# B&R Automation Studio project A2019059_Linka_Power_CP (part 30)

#### AtlasCopcoKomunikacia.st
```iecst
ACTION AtlasCopcoKomunikacia:

    M5_PrevodMomentu();
    M4_PrevodMomentu();
    M6_PrevodMomentu();

	//*********************************************************Skrutkovacka M5******************************************************************//
	//Vstupy z AtlasCopco do PLC//
    P2_Srobovanie.Skrutkovacka_M5.Stav_VysledokPotvrdeny:= P2_Srobovanie.PAR.M5_AtlasCopcoInputs[0].0;
    P2_Srobovanie.Skrutkovacka_M5.Stav_EmergencyStop:= P2_Srobovanie.PAR.M5_AtlasCopcoInputs[0].1;
    P2_Srobovanie.Skrutkovacka_M5.Stav_READY_to_START:= P2_Srobovanie.PAR.M5_AtlasCopcoInputs[0].2;
    P2_Srobovanie.Skrutkovacka_M5.Stav_MANUAL:= P2_Srobovanie.PAR.M5_AtlasCopcoInputs[0].3;
    P2_Srobovanie.Skrutkovacka_M5.Stav_UtahovanieUkoncene:= P2_Srobovanie.PAR.M5_AtlasCopcoInputs[0].4;
    P2_Srobovanie.Skrutkovacka_M5.Stav_VysledokUtahovania_NG:= P2_Srobovanie.PAR.M5_AtlasCopcoInputs[0].5;
    P2_Srobovanie.Skrutkovacka_M5.Stav_VysledokUtahovania_OK:= P2_Srobovanie.PAR.M5_AtlasCopcoInputs[0].6;
    P2_Srobovanie.Skrutkovacka_M5.Stav_SmerOtacania_VPRED:= P2_Srobovanie.PAR.M5_AtlasCopcoInputs[0].7;
    P2_Srobovanie.Skrutkovacka_M5.Stav_BUSY:= P2_Srobovanie.PAR.M5_AtlasCopcoInputs[0].8;
    P2_Srobovanie.Skrutkovacka_M5.Stav_ControlerSwitch_ON:= P2_Srobovanie.PAR.M5_AtlasCopcoInputs[0].9;
    P2_Srobovanie.Skrutkovacka_M5.Stav_Station_READY:= P2_Srobovanie.PAR.M5_AtlasCopcoInputs[0].10;
    P2_Srobovanie.Skrutkovacka_M5.Stav_NastrojPripojeny:= P2_Srobovanie.PAR.M5_AtlasCopcoInputs[0].11;
    P2_Srobovanie.Skrutkovacka_M5.Stav_NastrojUtahuje:= P2_Srobovanie.PAR.M5_AtlasCopcoInputs[0].12;

    //Výstupy z PLC do AtlasCopco//
    P2_Srobovanie.PAR.M5_AllasCopcoOutputs[0].0:= P2_Srobovanie.Skrutkovacka_M5.RESET_Poruchy;
    P2_Srobovanie.PAR.M5_AllasCopcoOutputs[0].1:= P2_Srobovanie.Skrutkovacka_M5.RESET_Vysledkov;
    P2_Srobovanie.PAR.M5_AllasCopcoOutputs[0].2:= P2_Srobovanie.Skrutkovacka_M5.START_Skrutkovania;
    P2_Srobovanie.PAR.M5_AllasCopcoOutputs[0].3:= P2_Srobovanie.Skrutkovacka_M5.START_Utahovania;

    //Dosiahnutý moment//
//    P2_Srobovanie.STAV.M5_DosiahnutyMoment.0:= P2_Srobovanie.PAR.M5_AtlasCopcoInputs[1].24;
//    P2_Srobovanie.STAV.M5_DosiahnutyMoment.1:= P2_Srobovanie.PAR.M5_AtlasCopcoInputs[1].25;
//    P2_Srobovanie.STAV.M5_DosiahnutyMoment.2:= P2_Srobovanie.PAR.M5_AtlasCopcoInputs[1].26;
//    P2_Srobovanie.STAV.M5_DosiahnutyMoment.3:= P2_Srobovanie.PAR.M5_AtlasCopcoInputs[1].27;
//    P2_Srobovanie.STAV.M5_DosiahnutyMoment.4:= P2_Srobovanie.PAR.M5_AtlasCopcoInputs[1].28;
//    P2_Srobovanie.STAV.M5_DosiahnutyMoment.5:= P2_Srobovanie.PAR.M5_AtlasCopcoInputs[1].29;
//    P2_Srobovanie.STAV.M5_DosiahnutyMoment.6:= P2_Srobovanie.PAR.M5_AtlasCopcoInputs[1].30;
//    P2_Srobovanie.STAV.M5_DosiahnutyMoment.7:= P2_Srobovanie.PAR.M5_AtlasCopcoInputs[1].31;
//    P2_Srobovanie.STAV.M5_DosiahnutyMoment.8:= P2_Srobovanie.PAR.M5_AtlasCopcoInputs[1].16;
//    P2_Srobovanie.STAV.M5_DosiahnutyMoment.9:= P2_Srobovanie.PAR.M5_AtlasCopcoInputs[1].17;
//    P2_Srobovanie.STAV.M5_DosiahnutyMoment.10:= P2_Srobovanie.PAR.M5_AtlasCopcoInputs[1].18;
//    P2_Srobovanie.STAV.M5_DosiahnutyMoment.11:= P2_Srobovanie.PAR.M5_AtlasCopcoInputs[1].19;
//    P2_Srobovanie.STAV.M5_DosiahnutyMoment.12:= P2_Srobovanie.PAR.M5_AtlasCopcoInputs[1].20;
//    P2_Srobovanie.STAV.M5_DosiahnutyMoment.13:= P2_Srobovanie.PAR.M5_AtlasCopcoInputs[1].21;
//    P2_Srobovanie.STAV.M5_DosiahnutyMoment.14:= P2_Srobovanie.PAR.M5_AtlasCopcoInputs[1].22;
//    P2_Srobovanie.STAV.M5_DosiahnutyMoment.15:= P2_Srobovanie.PAR.M5_AtlasCopcoInputs[1].23;
//    P2_Srobovanie.STAV.M5_DosiahnutyMoment.16:= P2_Srobovanie.PAR.M5_AtlasCopcoInputs[1].8;
//    P2_Srobovanie.STAV.M5_DosiahnutyMoment.17:= P2_Srobovanie.PAR.M5_AtlasCopcoInputs[1].9;
//    P2_Srobovanie.STAV.M5_DosiahnutyMoment.18:= P2_Srobovanie.PAR.M5_AtlasCopcoInputs[1].10;
//    P2_Srobovanie.STAV.M5_DosiahnutyMoment.19:= P2_Srobovanie.PAR.M5_AtlasCopcoInputs[1].11;
//    P2_Srobovanie.STAV.M5_DosiahnutyMoment.20:= P2_Srobovanie.PAR.M5_AtlasCopcoInputs[1].12;
//    P2_Srobovanie.STAV.M5_DosiahnutyMoment.21:= P2_Srobovanie.PAR.M5_AtlasCopcoInputs[1].13;
//    P2_Srobovanie.STAV.M5_DosiahnutyMoment.22:= P2_Srobovanie.PAR.M5_AtlasCopcoInputs[1].14;
//    P2_Srobovanie.STAV.M5_DosiahnutyMoment.23:= P2_Srobovanie.PAR.M5_AtlasCopcoInputs[1].15;
//    P2_Srobovanie.STAV.M5_DosiahnutyMoment.24:= P2_Srobovanie.PAR.M5_AtlasCopcoInputs[1].0;
//    P2_Srobovanie.STAV.M5_DosiahnutyMoment.25:= P2_Srobovanie.PAR.M5_AtlasCopcoInputs[1].1;
//    P2_Srobovanie.STAV.M5_DosiahnutyMoment.26:= P2_Srobovanie.PAR.M5_AtlasCopcoInputs[1].2;
//    P2_Srobovanie.STAV.M5_DosiahnutyMoment.27:= P2_Srobovanie.PAR.M5_AtlasCopcoInputs[1].3;
//    P2_Srobovanie.STAV.M5_DosiahnutyMoment.28:= P2_Srobovanie.PAR.M5_AtlasCopcoInputs[1].4;
//    P2_Srobovanie.STAV.M5_DosiahnutyMoment.29:= P2_Srobovanie.PAR.M5_AtlasCopcoInputs[1].5;
//    P2_Srobovanie.STAV.M5_DosiahnutyMoment.30:= P2_Srobovanie.PAR.M5_AtlasCopcoInputs[1].6;
//    P2_Srobovanie.STAV.M5_DosiahnutyMoment.31:= P2_Srobovanie.PAR.M5_AtlasCopcoInputs[1].7;
//    M5_DosiahnutyMoment_REAL:= UDINT_TO_REAL(P2_Srobovanie.STAV.M5_DosiahnutyMoment);
//    IF M5_DosiahnutyMoment_REAL > 0 THEN
//        P2_Srobovanie.STAV.M5_DosiahnutyMoment_REAL:= M5_DosiahnutyMoment_REAL/100;
//    ELSE
//        P2_Srobovanie.STAV.M5_DosiahnutyMoment_REAL:= 0.0;
//    END_IF

    M5_PrevodMomentu.AtlasAktualnyMoment:=P2_Srobovanie.PAR.M5_AtlasCopcoInputs[1];
    P2_Srobovanie.STAV.M5_DosiahnutyMoment_REAL:=M5_PrevodMomentu.AktualnyMoment;

    //Moment - Tolerancia MAX//
//    P2_Srobovanie.STAV.M5_Moment_ToleranciaMAX.0:= P2_Srobovanie.PAR.M5_AtlasCopcoInputs[3].24;
//    P2_Srobovanie.STAV.M5_Moment_ToleranciaMAX.1:= P2_Srobovanie.PAR.M5_AtlasCopcoInputs[3].25;
//    P2_Srobovanie.STAV.M5_Moment_ToleranciaMAX.2:= P2_Srobovanie.PAR.M5_AtlasCopcoInputs[3].26;
//    P2_Srobovanie.STAV.M5_Moment_ToleranciaMAX.3:= P2_Srobovanie.PAR.M5_AtlasCopcoInputs[3].27;
//    P2_Srobovanie.STAV.M5_Moment_ToleranciaMAX.4:= P2_Srobovanie.PAR.M5_AtlasCopcoInputs[3].28;
//    P2_Srobovanie.STAV.M5_Moment_ToleranciaMAX.5:= P2_Srobovanie.PAR.M5_AtlasCopcoInputs[3].29;
//    P2_Srobovanie.STAV.M5_Moment_ToleranciaMAX.6:= P2_Srobovanie.PAR.M5_AtlasCopcoInputs[3].30;
//    P2_Srobovanie.STAV.M5_Moment_ToleranciaMAX.7:= P2_Srobovanie.PAR.M5_AtlasCopcoInputs[3].31;
//    P2_Srobovanie.STAV.M5_Moment_ToleranciaMAX.8:= P2_Srobovanie.PAR.M5_AtlasCopcoInputs[3].16;
//    P2_Srobovanie.STAV.M5_Moment_ToleranciaMAX.9:= P2_Srobovanie.PAR.M5_AtlasCopcoInputs[3].17;
//    P2_Srobovanie.STAV.M5_Moment_ToleranciaMAX.10:= P2_Srobovanie.PAR.M5_AtlasCopcoInputs[3].18;
//    P2_Srobovanie.STAV.M5_Moment_ToleranciaMAX.11:= P2_Srobovanie.PAR.M5_AtlasCopcoInputs[3].19;
//    P2_Srobovanie.STAV.M5_Moment_ToleranciaMAX.12:= P2_Srobovanie.PAR.M5_AtlasCopcoInputs[3].20;
//    P2_Srobovanie.STAV.M5_Moment_ToleranciaMAX.13:= P2_Srobovanie.PAR.M5_AtlasCopcoInputs[3].21;
//    P2_Srobovanie.STAV.M5_Moment_ToleranciaMAX.14:= P2_Srobovanie.PAR.M5_AtlasCopcoInputs[3].22;
//    P2_Srobovanie.STAV.M5_Moment_ToleranciaMAX.15:= P2_Srobovanie.PAR.M5_AtlasCopcoInputs[3].23;
//    P2_Srobovanie.STAV.M5_Moment_ToleranciaMAX.16:= P2_Srobovanie.PAR.M5_AtlasCopcoInputs[3].8;
//    P2_Srobovanie.STAV.M5_Moment_ToleranciaMAX.17:= P2_Srobovanie.PAR.M5_AtlasCopcoInputs[3].9;
//    P2_Srobovanie.STAV.M5_Moment_ToleranciaMAX.18:= P2_Srobovanie.PAR.M5_AtlasCopcoInputs[3].10;
//    P2_Srobovanie.STAV.M5_Moment_ToleranciaMAX.19:= P2_Srobovanie.PAR.M5_AtlasCopcoInputs[3].11;
//    P2_Srobovanie.STAV.M5_Moment_ToleranciaMAX.20:= P2_Srobovanie.PAR.M5_AtlasCopcoInputs[3].12;
//    P2_Srobovanie.STAV.M5_Moment_ToleranciaMAX.21:= P2_Srobovanie.PAR.M5_AtlasCopcoInputs[3].13;
//    P2_Srobovanie.STAV.M5_Moment_ToleranciaMAX.22:= P2_Srobovanie.PAR.M5_AtlasCopcoInputs[3].14;
//    P2_Srobovanie.STAV.M5_Moment_ToleranciaMAX.23:= P2_Srobovanie.PAR.M5_AtlasCopcoInputs[3].15;
//    P2_Srobovanie.STAV.M5_Moment_ToleranciaMAX.24:= P2_Srobovanie.PAR.M5_AtlasCopcoInputs[3].0;
//    P2_Srobovanie.STAV.M5_Moment_ToleranciaMAX.25:= P2_Srobovanie.PAR.M5_AtlasCopcoInputs[3].1;
//    P2_Srobovanie.STAV.M5_Moment_ToleranciaMAX.26:= P2_Srobovanie.PAR.M5_AtlasCopcoInputs[3].2;
//    P2_Srobovanie.STAV.M5_Moment_ToleranciaMAX.27:= P2_Srobovanie.PAR.M5_AtlasCopcoInputs[3].3;
//    P2_Srobovanie.STAV.M5_Moment_ToleranciaMAX.28:= P2_Srobovanie.PAR.M5_AtlasCopcoInputs[3].4;
//    P2_Srobovanie.STAV.M5_Moment_ToleranciaMAX.29:= P2_Srobovanie.PAR.M5_AtlasCopcoInputs[3].5;
//    P2_Srobovanie.STAV.M5_Moment_ToleranciaMAX.30:= P2_Srobovanie.PAR.M5_AtlasCopcoInputs[3].6;
//    P2_Srobovanie.STAV.M5_Moment_ToleranciaMAX.31:= P2_Srobovanie.PAR.M5_AtlasCopcoInputs[3].7;
//    M5_Moment_ToleranciaMAX_REAL:= UDINT_TO_REAL(P2_Srobovanie.STAV.M5_Moment_ToleranciaMAX);
//    IF M5_Moment_ToleranciaMAX_REAL > 0 THEN
//        P2_Srobovanie.STAV.M5_Moment_ToleranciaMAX_REAL:= M5_Moment_ToleranciaMAX_REAL/100;
//    ELSE
//        P2_Srobovanie.STAV.M5_Moment_ToleranciaMAX_REAL:= 0.0;
//    END_IF

    M5_PrevodMomentu.AtlasMaximalnaTolerancia:=P2_Srobovanie.PAR.M5_AtlasCopcoInputs[3];
    P2_Srobovanie.STAV.M5_Moment_ToleranciaMAX_REAL:=M5_PrevodMomentu.ToleranciaMAX;

    //Moment - Tolerancia MIN//
//    P2_Srobovanie.STAV.M5_Moment_ToleranciaMIN.0:= P2_Srobovanie.PAR.M5_AtlasCopcoInputs[4].24;
//    P2_Srobovanie.STAV.M5_Moment_ToleranciaMIN.1:= P2_Srobovanie.PAR.M5_AtlasCopcoInputs[4].25;
//    P2_Srobovanie.STAV.M5_Moment_ToleranciaMIN.2:= P2_Srobovanie.PAR.M5_AtlasCopcoInputs[4].26;
//    P2_Srobovanie.STAV.M5_Moment_ToleranciaMIN.3:= P2_Srobovanie.PAR.M5_AtlasCopcoInputs[4].27;
//    P2_Srobovanie.STAV.M5_Moment_ToleranciaMIN.4:= P2_Srobovanie.PAR.M5_AtlasCopcoInputs[4].28;
//    P2_Srobovanie.STAV.M5_Moment_ToleranciaMIN.5:= P2_Srobovanie.PAR.M5_AtlasCopcoInputs[4].29;
//    P2_Srobovanie.STAV.M5_Moment_ToleranciaMIN.6:= P2_Srobovanie.PAR.M5_AtlasCopcoInputs[4].30;
//    P2_Srobovanie.STAV.M5_Moment_ToleranciaMIN.7:= P2_Srobovanie.PAR.M5_AtlasCopcoInputs[4].31;
//    P2_Srobovanie.STAV.M5_Moment_ToleranciaMIN.8:= P2_Srobovanie.PAR.M5_AtlasCopcoInputs[4].16;
//    P2_Srobovanie.STAV.M5_Moment_ToleranciaMIN.9:= P2_Srobovanie.PAR.M5_AtlasCopcoInputs[4].17;
//    P2_Srobovanie.STAV.M5_Moment_ToleranciaMIN.10:= P2_Srobovanie.PAR.M5_AtlasCopcoInputs[4].18;
//    P2_Srobovanie.STAV.M5_Moment_ToleranciaMIN.11:= P2_Srobovanie.PAR.M5_AtlasCopcoInputs[4].19;
//    P2_Srobovanie.STAV.M5_Moment_ToleranciaMIN.12:= P2_Srobovanie.PAR.M5_AtlasCopcoInputs[4].20;
//    P2_Srobovanie.STAV.M5_Moment_ToleranciaMIN.13:= P2_Srobovanie.PAR.M5_AtlasCopcoInputs[4].21;
//    P2_Srobovanie.STAV.M5_Moment_ToleranciaMIN.14:= P2_Srobovanie.PAR.M5_AtlasCopcoInputs[4].22;
//    P2_Srobovanie.STAV.M5_Moment_ToleranciaMIN.15:= P2_Srobovanie.PAR.M5_AtlasCopcoInputs[4].23;
//    P2_Srobovanie.STAV.M5_Moment_ToleranciaMIN.16:= P2_Srobovanie.PAR.M5_AtlasCopcoInputs[4].8;
//    P2_Srobovanie.STAV.M5_Moment_ToleranciaMIN.17:= P2_Srobovanie.PAR.M5_AtlasCopcoInputs[4].9;
//    P2_Srobovanie.STAV.M5_Moment_ToleranciaMIN.18:= P2_Srobovanie.PAR.M5_AtlasCopcoInputs[4].10;
//    P2_Srobovanie.STAV.M5_Moment_ToleranciaMIN.19:= P2_Srobovanie.PAR.M5_AtlasCopcoInputs[4].11;
//    P2_Srobovanie.STAV.M5_Moment_ToleranciaMIN.20:= P2_Srobovanie.PAR.M5_AtlasCopcoInputs[4].12;
//    P2_Srobovanie.STAV.M5_Moment_ToleranciaMIN.21:= P2_Srobovanie.PAR.M5_AtlasCopcoInputs[4].13;
//    P2_Srobovanie.STAV.M5_Moment_ToleranciaMIN.22:= P2_Srobovanie.PAR.M5_AtlasCopcoInputs[4].14;
//    P2_Srobovanie.STAV.M5_Moment_ToleranciaMIN.23:= P2_Srobovanie.PAR.M5_AtlasCopcoInputs[4].15;
//    P2_Srobovanie.STAV.M5_Moment_ToleranciaMIN.24:= P2_Srobovanie.PAR.M5_AtlasCopcoInputs[4].0;
//    P2_Srobovanie.STAV.M5_Moment_ToleranciaMIN.25:= P2_Srobovanie.PAR.M5_AtlasCopcoInputs[4].1;
//    P2_Srobovanie.STAV.M5_Moment_ToleranciaMIN.26:= P2_Srobovanie.PAR.M5_AtlasCopcoInputs[4].2;
//    P2_Srobovanie.STAV.M5_Moment_ToleranciaMIN.27:= P2_Srobovanie.PAR.M5_AtlasCopcoInputs[4].3;
//    P2_Srobovanie.STAV.M5_Moment_ToleranciaMIN.28:= P2_Srobovanie.PAR.M5_AtlasCopcoInputs[4].4;
//    P2_Srobovanie.STAV.M5_Moment_ToleranciaMIN.29:= P2_Srobovanie.PAR.M5_AtlasCopcoInputs[4].5;
//    P2_Srobovanie.STAV.M5_Moment_ToleranciaMIN.30:= P2_Srobovanie.PAR.M5_AtlasCopcoInputs[4].6;
//    P2_Srobovanie.STAV.M5_Moment_ToleranciaMIN.31:= P2_Srobovanie.PAR.M5_AtlasCopcoInputs[4].7;
//    M5_Moment_ToleranciaMIN_REAL:= UDINT_TO_REAL(P2_Srobovanie.STAV.M5_Moment_ToleranciaMIN);
//    IF M5_Moment_ToleranciaMIN_REAL > 0 THEN
//        P2_Srobovanie.STAV.M5_Moment_ToleranciaMIN_REAL:= M5_Moment_ToleranciaMIN_REAL /100;
//    ELSE
//        P2_Srobovanie.STAV.M5_Moment_ToleranciaMIN_REAL:= 0.0;
    //    END_IF

    M5_PrevodMomentu.AtlasMinimalnaTolerancia:=P2_Srobovanie.PAR.M5_AtlasCopcoInputs[4];
    P2_Srobovanie.STAV.M5_Moment_ToleranciaMIN_REAL:=M5_PrevodMomentu.ToleranciaMIN;

    //Dosiahnutý úhol//
    P2_Srobovanie.STAV.M5_DosiahnutyUhol.0:= P2_Srobovanie.PAR.M5_AtlasCopcoInputs[0].24;
    P2_Srobovanie.STAV.M5_DosiahnutyUhol.1:= P2_Srobovanie.PAR.M5_AtlasCopcoInputs[0].25;
    P2_Srobovanie.STAV.M5_DosiahnutyUhol.2:= P2_Srobovanie.PAR.M5_AtlasCopcoInputs[0].26;
    P2_Srobovanie.STAV.M5_DosiahnutyUhol.3:= P2_Srobovanie.PAR.M5_AtlasCopcoInputs[0].27;
    P2_Srobovanie.STAV.M5_DosiahnutyUhol.4:= P2_Srobovanie.PAR.M5_AtlasCopcoInputs[0].28;
    P2_Srobovanie.STAV.M5_DosiahnutyUhol.5:= P2_Srobovanie.PAR.M5_AtlasCopcoInputs[0].29;
    P2_Srobovanie.STAV.M5_DosiahnutyUhol.6:= P2_Srobovanie.PAR.M5_AtlasCopcoInputs[0].30;
    P2_Srobovanie.STAV.M5_DosiahnutyUhol.7:= P2_Srobovanie.PAR.M5_AtlasCopcoInputs[0].31;
    P2_Srobovanie.STAV.M5_DosiahnutyUhol.8:= P2_Srobovanie.PAR.M5_AtlasCopcoInputs[0].16;
    P2_Srobovanie.STAV.M5_DosiahnutyUhol.9:= P2_Srobovanie.PAR.M5_AtlasCopcoInputs[0].17;
    P2_Srobovanie.STAV.M5_DosiahnutyUhol.10:= P2_Srobovanie.PAR.M5_AtlasCopcoInputs[0].18;
    P2_Srobovanie.STAV.M5_DosiahnutyUhol.11:= P2_Srobovanie.PAR.M5_AtlasCopcoInputs[0].19;
    P2_Srobovanie.STAV.M5_DosiahnutyUhol.12:= P2_Srobovanie.PAR.M5_AtlasCopcoInputs[0].20;
    P2_Srobovanie.STAV.M5_DosiahnutyUhol.13:= P2_Srobovanie.PAR.M5_AtlasCopcoInputs[0].21;
    P2_Srobovanie.STAV.M5_DosiahnutyUhol.14:= P2_Srobovanie.PAR.M5_AtlasCopcoInputs[0].22;
    P2_Srobovanie.STAV.M5_DosiahnutyUhol.15:= P2_Srobovanie.PAR.M5_AtlasCopcoInputs[0].23;

    //Uhol - Tolerancia MAX//
    P2_Srobovanie.STAV.M5_Uhol_ToleranciaMAX.0:= P2_Srobovanie.PAR.M5_AtlasCopcoInputs[2].8;
    P2_Srobovanie.STAV.M5_Uhol_ToleranciaMAX.1:= P2_Srobovanie.PAR.M5_AtlasCopcoInputs[2].9;
    P2_Srobovanie.STAV.M5_Uhol_ToleranciaMAX.2:= P2_Srobovanie.PAR.M5_AtlasCopcoInputs[2].10;
    P2_Srobovanie.STAV.M5_Uhol_ToleranciaMAX.3:= P2_Srobovanie.PAR.M5_AtlasCopcoInputs[2].11;
    P2_Srobovanie.STAV.M5_Uhol_ToleranciaMAX.4:= P2_Srobovanie.PAR.M5_AtlasCopcoInputs[2].12;
    P2_Srobovanie.STAV.M5_Uhol_ToleranciaMAX.5:= P2_Srobovanie.PAR.M5_AtlasCopcoInputs[2].13;
    P2_Srobovanie.STAV.M5_Uhol_ToleranciaMAX.6:= P2_Srobovanie.PAR.M5_AtlasCopcoInputs[2].14;
    P2_Srobovanie.STAV.M5_Uhol_ToleranciaMAX.7:= P2_Srobovanie.PAR.M5_AtlasCopcoInputs[2].15;
    P2_Srobovanie.STAV.M5_Uhol_ToleranciaMAX.8:= P2_Srobovanie.PAR.M5_AtlasCopcoInputs[2].0;
    P2_Srobovanie.STAV.M5_Uhol_ToleranciaMAX.9:= P2_Srobovanie.PAR.M5_AtlasCopcoInputs[2].1;
    P2_Srobovanie.STAV.M5_Uhol_ToleranciaMAX.10:= P2_Srobovanie.PAR.M5_AtlasCopcoInputs[2].2;
    P2_Srobovanie.STAV.M5_Uhol_ToleranciaMAX.11:= P2_Srobovanie.PAR.M5_AtlasCopcoInputs[2].3;
    P2_Srobovanie.STAV.M5_Uhol_ToleranciaMAX.12:= P2_Srobovanie.PAR.M5_AtlasCopcoInputs[2].4;
    P2_Srobovanie.STAV.M5_Uhol_ToleranciaMAX.13:= P2_Srobovanie.PAR.M5_AtlasCopcoInputs[2].5;
    P2_Srobovanie.STAV.M5_Uhol_ToleranciaMAX.14:= P2_Srobovanie.PAR.M5_AtlasCopcoInputs[2].6;
    P2_Srobovanie.STAV.M5_Uhol_ToleranciaMAX.15:= P2_Srobovanie.PAR.M5_AtlasCopcoInputs[2].7;

    //Uhol - Tolerancia MIN//
    P2_Srobovanie.STAV.M5_Uhol_ToleranciaMIN.0:= P2_Srobovanie.PAR.M5_AtlasCopcoInputs[2].24;
    P2_Srobovanie.STAV.M5_Uhol_ToleranciaMIN.1:= P2_Srobovanie.PAR.M5_AtlasCopcoInputs[2].25;
    P2_Srobovanie.STAV.M5_Uhol_ToleranciaMIN.2:= P2_Srobovanie.PAR.M5_AtlasCopcoInputs[2].26;
    P2_Srobovanie.STAV.M5_Uhol_ToleranciaMIN.3:= P2_Srobovanie.PAR.M5_AtlasCopcoInputs[2].27;
    P2_Srobovanie.STAV.M5_Uhol_ToleranciaMIN.4:= P2_Srobovanie.PAR.M5_AtlasCopcoInputs[2].28;
    P2_Srobovanie.STAV.M5_Uhol_ToleranciaMIN.5:= P2_Srobovanie.PAR.M5_AtlasCopcoInputs[2].29;
    P2_Srobovanie.STAV.M5_Uhol_ToleranciaMIN.6:= P2_Srobovanie.PAR.M5_AtlasCopcoInputs[2].30;
    P2_Srobovanie.STAV.M5_Uhol_ToleranciaMIN.7:= P2_Srobovanie.PAR.M5_AtlasCopcoInputs[2].31;
    P2_Srobovanie.STAV.M5_Uhol_ToleranciaMIN.8:= P2_Srobovanie.PAR.M5_AtlasCopcoInputs[2].16;
    P2_Srobovanie.STAV.M5_Uhol_ToleranciaMIN.9:= P2_Srobovanie.PAR.M5_AtlasCopcoInputs[2].17;
    P2_Srobovanie.STAV.M5_Uhol_ToleranciaMIN.10:= P2_Srobovanie.PAR.M5_AtlasCopcoInputs[2].18;
    P2_Srobovanie.STAV.M5_Uhol_ToleranciaMIN.11:= P2_Srobovanie.PAR.M5_AtlasCopcoInputs[2].19;
    P2_Srobovanie.STAV.M5_Uhol_ToleranciaMIN.12:= P2_Srobovanie.PAR.M5_AtlasCopcoInputs[2].20;
    P2_Srobovanie.STAV.M5_Uhol_ToleranciaMIN.13:= P2_Srobovanie.PAR.M5_AtlasCopcoInputs[2].21;
    P2_Srobovanie.STAV.M5_Uhol_ToleranciaMIN.14:= P2_Srobovanie.PAR.M5_AtlasCopcoInputs[2].22;
    P2_Srobovanie.STAV.M5_Uhol_ToleranciaMIN.15:= P2_Srobovanie.PAR.M5_AtlasCopcoInputs[2].23;

    //*****************************************************************************Skrutkovacka M4*************************************************************//
    //Vstupy z AtlasCopco do PLC//
    P2_Srobovanie.Skrutkovacka_M4.Stav_VysledokPotvrdeny:= P2_Srobovanie.PAR.M4_AtlasCopcoInputs[0].0;
    P2_Srobovanie.Skrutkovacka_M4.Stav_EmergencyStop:= P2_Srobovanie.PAR.M4_AtlasCopcoInputs[0].1;
    P2_Srobovanie.Skrutkovacka_M4.Stav_READY_to_START:= P2_Srobovanie.PAR.M4_AtlasCopcoInputs[0].2;
    P2_Srobovanie.Skrutkovacka_M4.Stav_MANUAL:= P2_Srobovanie.PAR.M4_AtlasCopcoInputs[0].3;
    P2_Srobovanie.Skrutkovacka_M4.Stav_UtahovanieUkoncene:= P2_Srobovanie.PAR.M4_AtlasCopcoInputs[0].4;
    P2_Srobovanie.Skrutkovacka_M4.Stav_VysledokUtahovania_NG:= P2_Srobovanie.PAR.M4_AtlasCopcoInputs[0].5;
    P2_Srobovanie.Skrutkovacka_M4.Stav_VysledokUtahovania_OK:= P2_Srobovanie.PAR.M4_AtlasCopcoInputs[0].6;
    P2_Srobovanie.Skrutkovacka_M4.Stav_SmerOtacania_VPRED:= P2_Srobovanie.PAR.M4_AtlasCopcoInputs[0].7;
    P2_Srobovanie.Skrutkovacka_M4.Stav_BUSY:= P2_Srobovanie.PAR.M4_AtlasCopcoInputs[0].8;
    P2_Srobovanie.Skrutkovacka_M4.Stav_ControlerSwitch_ON:= P2_Srobovanie.PAR.M4_AtlasCopcoInputs[0].9;
    P2_Srobovanie.Skrutkovacka_M4.Stav_Station_READY:= P2_Srobovanie.PAR.M4_AtlasCopcoInputs[0].10;
    P2_Srobovanie.Skrutkovacka_M4.Stav_NastrojPripojeny:= P2_Srobovanie.PAR.M4_AtlasCopcoInputs[0].11;
    P2_Srobovanie.Skrutkovacka_M4.Stav_NastrojUtahuje:= P2_Srobovanie.PAR.M4_AtlasCopcoInputs[0].12;

    //Výstupy z PLC do AtlasCopco//
    P2_Srobovanie.PAR.M4_AllasCopcoOutputs[0].0:= P2_Srobovanie.Skrutkovacka_M4.RESET_Poruchy;
    P2_Srobovanie.PAR.M4_AllasCopcoOutputs[0].1:= P2_Srobovanie.Skrutkovacka_M4.RESET_Vysledkov;
    P2_Srobovanie.PAR.M4_AllasCopcoOutputs[0].2:= P2_Srobovanie.Skrutkovacka_M4.START_Skrutkovania;
    P2_Srobovanie.PAR.M4_AllasCopcoOutputs[0].3:= P2_Srobovanie.Skrutkovacka_M4.START_Utahovania;

    //Dosiahnutý moment//
//    P2_Srobovanie.STAV.M4_DosiahnutyMoment.0:= P2_Srobovanie.PAR.M4_AtlasCopcoInputs[1].24;
//    P2_Srobovanie.STAV.M4_DosiahnutyMoment.1:= P2_Srobovanie.PAR.M4_AtlasCopcoInputs[1].25;
//    P2_Srobovanie.STAV.M4_DosiahnutyMoment.2:= P2_Srobovanie.PAR.M4_AtlasCopcoInputs[1].26;
//    P2_Srobovanie.STAV.M4_DosiahnutyMoment.3:= P2_Srobovanie.PAR.M4_AtlasCopcoInputs[1].27;
//    P2_Srobovanie.STAV.M4_DosiahnutyMoment.4:= P2_Srobovanie.PAR.M4_AtlasCopcoInputs[1].28;
//    P2_Srobovanie.STAV.M4_DosiahnutyMoment.5:= P2_Srobovanie.PAR.M4_AtlasCopcoInputs[1].29;
//    P2_Srobovanie.STAV.M4_DosiahnutyMoment.6:= P2_Srobovanie.PAR.M4_AtlasCopcoInputs[1].30;
//    P2_Srobovanie.STAV.M4_DosiahnutyMoment.7:= P2_Srobovanie.PAR.M4_AtlasCopcoInputs[1].31;
//    P2_Srobovanie.STAV.M4_DosiahnutyMoment.8:= P2_Srobovanie.PAR.M4_AtlasCopcoInputs[1].16;
//    P2_Srobovanie.STAV.M4_DosiahnutyMoment.9:= P2_Srobovanie.PAR.M4_AtlasCopcoInputs[1].17;
//    P2_Srobovanie.STAV.M4_DosiahnutyMoment.10:= P2_Srobovanie.PAR.M4_AtlasCopcoInputs[1].18;
//    P2_Srobovanie.STAV.M4_DosiahnutyMoment.11:= P2_Srobovanie.PAR.M4_AtlasCopcoInputs[1].19;
//    P2_Srobovanie.STAV.M4_DosiahnutyMoment.12:= P2_Srobovanie.PAR.M4_AtlasCopcoInputs[1].20;
//    P2_Srobovanie.STAV.M4_DosiahnutyMoment.13:= P2_Srobovanie.PAR.M4_AtlasCopcoInputs[1].21;
//    P2_Srobovanie.STAV.M4_DosiahnutyMoment.14:= P2_Srobovanie.PAR.M4_AtlasCopcoInputs[1].22;
//    P2_Srobovanie.STAV.M4_DosiahnutyMoment.15:= P2_Srobovanie.PAR.M4_AtlasCopcoInputs[1].23;
//    P2_Srobovanie.STAV.M4_DosiahnutyMoment.16:= P2_Srobovanie.PAR.M4_AtlasCopcoInputs[1].8;
//    P2_Srobovanie.STAV.M4_DosiahnutyMoment.17:= P2_Srobovanie.PAR.M4_AtlasCopcoInputs[1].9;
//    P2_Srobovanie.STAV.M4_DosiahnutyMoment.18:= P2_Srobovanie.PAR.M4_AtlasCopcoInputs[1].10;
//    P2_Srobovanie.STAV.M4_DosiahnutyMoment.19:= P2_Srobovanie.PAR.M4_AtlasCopcoInputs[1].11;
//    P2_Srobovanie.STAV.M4_DosiahnutyMoment.20:= P2_Srobovanie.PAR.M4_AtlasCopcoInputs[1].12;
//    P2_Srobovanie.STAV.M4_DosiahnutyMoment.21:= P2_Srobovanie.PAR.M4_AtlasCopcoInputs[1].13;
//    P2_Srobovanie.STAV.M4_DosiahnutyMoment.22:= P2_Srobovanie.PAR.M4_AtlasCopcoInputs[1].14;
//    P2_Srobovanie.STAV.M4_DosiahnutyMoment.23:= P2_Srobovanie.PAR.M4_AtlasCopcoInputs[1].15;
//    P2_Srobovanie.STAV.M4_DosiahnutyMoment.24:= P2_Srobovanie.PAR.M4_AtlasCopcoInputs[1].0;
//    P2_Srobovanie.STAV.M4_DosiahnutyMoment.25:= P2_Srobovanie.PAR.M4_AtlasCopcoInputs[1].1;
//    P2_Srobovanie.STAV.M4_DosiahnutyMoment.26:= P2_Srobovanie.PAR.M4_AtlasCopcoInputs[1].2;
//    P2_Srobovanie.STAV.M4_DosiahnutyMoment.27:= P2_Srobovanie.PAR.M4_AtlasCopcoInputs[1].3;
//    P2_Srobovanie.STAV.M4_DosiahnutyMoment.28:= P2_Srobovanie.PAR.M4_AtlasCopcoInputs[1].4;
//    P2_Srobovanie.STAV.M4_DosiahnutyMoment.29:= P2_Srobovanie.PAR.M4_AtlasCopcoInputs[1].5;
//    P2_Srobovanie.STAV.M4_DosiahnutyMoment.30:= P2_Srobovanie.PAR.M4_AtlasCopcoInputs[1].6;
//    P2_Srobovanie.STAV.M4_DosiahnutyMoment.31:= P2_Srobovanie.PAR.M4_AtlasCopcoInputs[1].7;
//    M4_DosiahnutyMoment_REAL:= UDINT_TO_REAL(P2_Srobovanie.STAV.M4_DosiahnutyMoment);
//    IF M4_DosiahnutyMoment_REAL > 0 THEN
//      P2_Srobovanie.STAV.M4_DosiahnutyMoment_REAL:= (M4_DosiahnutyMoment_REAL*2.1)/131082;
//    ELSE
//        P2_Srobovanie.STAV.M4_DosiahnutyMoment_REAL:= 0.0;
//    END_IF
//    (*P2_Srobovanie.STAV.M4_DosiahnutyMoment_REAL:= M4_DosiahnutyMoment_REAL/100;*)

    M4_PrevodMomentu.AtlasAktualnyMoment:=P2_Srobovanie.PAR.M4_AtlasCopcoInputs[1];
    P2_Srobovanie.STAV.M4_DosiahnutyMoment_REAL:=M4_PrevodMomentu.AktualnyMoment;

    //Moment - Tolerancia MAX//
//    P2_Srobovanie.STAV.M4_Moment_ToleranciaMAX.0:= P2_Srobovanie.PAR.M4_AtlasCopcoInputs[3].24;
//    P2_Srobovanie.STAV.M4_Moment_ToleranciaMAX.1:= P2_Srobovanie.PAR.M4_AtlasCopcoInputs[3].25;
//    P2_Srobovanie.STAV.M4_Moment_ToleranciaMAX.2:= P2_Srobovanie.PAR.M4_AtlasCopcoInputs[3].26;
//    P2_Srobovanie.STAV.M4_Moment_ToleranciaMAX.3:= P2_Srobovanie.PAR.M4_AtlasCopcoInputs[3].27;
//    P2_Srobovanie.STAV.M4_Moment_ToleranciaMAX.4:= P2_Srobovanie.PAR.M4_AtlasCopcoInputs[3].28;
//    P2_Srobovanie.STAV.M4_Moment_ToleranciaMAX.5:= P2_Srobovanie.PAR.M4_AtlasCopcoInputs[3].29;
//    P2_Srobovanie.STAV.M4_Moment_ToleranciaMAX.6:= P2_Srobovanie.PAR.M4_AtlasCopcoInputs[3].30;
//    P2_Srobovanie.STAV.M4_Moment_ToleranciaMAX.7:= P2_Srobovanie.PAR.M4_AtlasCopcoInputs[3].31;
//    P2_Srobovanie.STAV.M4_Moment_ToleranciaMAX.8:= P2_Srobovanie.PAR.M4_AtlasCopcoInputs[3].16;
//    P2_Srobovanie.STAV.M4_Moment_ToleranciaMAX.9:= P2_Srobovanie.PAR.M4_AtlasCopcoInputs[3].17;
//    P2_Srobovanie.STAV.M4_Moment_ToleranciaMAX.10:= P2_Srobovanie.PAR.M4_AtlasCopcoInputs[3].18;
//    P2_Srobovanie.STAV.M4_Moment_ToleranciaMAX.11:= P2_Srobovanie.PAR.M4_AtlasCopcoInputs[3].19;
//    P2_Srobovanie.STAV.M4_Moment_ToleranciaMAX.12:= P2_Srobovanie.PAR.M4_AtlasCopcoInputs[3].20;
//    P2_Srobovanie.STAV.M4_Moment_ToleranciaMAX.13:= P2_Srobovanie.PAR.M4_AtlasCopcoInputs[3].21;
//    P2_Srobovanie.STAV.M4_Moment_ToleranciaMAX.14:= P2_Srobovanie.PAR.M4_AtlasCopcoInputs[3].22;
//    P2_Srobovanie.STAV.M4_Moment_ToleranciaMAX.15:= P2_Srobovanie.PAR.M4_AtlasCopcoInputs[3].23;
//    P2_Srobovanie.STAV.M4_Moment_ToleranciaMAX.16:= P2_Srobovanie.PAR.M4_AtlasCopcoInputs[3].8;
//    P2_Srobovanie.STAV.M4_Moment_ToleranciaMAX.17:= P2_Srobovanie.PAR.M4_AtlasCopcoInputs[3].9;
//    P2_Srobovanie.STAV.M4_Moment_ToleranciaMAX.18:= P2_Srobovanie.PAR.M4_AtlasCopcoInputs[3].10;
//    P2_Srobovanie.STAV.M4_Moment_ToleranciaMAX.19:= P2_Srobovanie.PAR.M4_AtlasCopcoInputs[3].11;
//    P2_Srobovanie.STAV.M4_Moment_ToleranciaMAX.20:= P2_Srobovanie.PAR.M4_AtlasCopcoInputs[3].12;
//    P2_Srobovanie.STAV.M4_Moment_ToleranciaMAX.21:= P2_Srobovanie.PAR.M4_AtlasCopcoInputs[3].13;
//    P2_Srobovanie.STAV.M4_Moment_ToleranciaMAX.22:= P2_Srobovanie.PAR.M4_AtlasCopcoInputs[3].14;
//    P2_Srobovanie.STAV.M4_Moment_ToleranciaMAX.23:= P2_Srobovanie.PAR.M4_AtlasCopcoInputs[3].15;
//    P2_Srobovanie.STAV.M4_Moment_ToleranciaMAX.24:= P2_Srobovanie.PAR.M4_AtlasCopcoInputs[3].0;
//    P2_Srobovanie.STAV.M4_Moment_ToleranciaMAX.25:= P2_Srobovanie.PAR.M4_AtlasCopcoInputs[3].1;
//    P2_Srobovanie.STAV.M4_Moment_ToleranciaMAX.26:= P2_Srobovanie.PAR.M4_AtlasCopcoInputs[3].2;
//    P2_Srobovanie.STAV.M4_Moment_ToleranciaMAX.27:= P2_Srobovanie.PAR.M4_AtlasCopcoInputs[3].3;
//    P2_Srobovanie.STAV.M4_Moment_ToleranciaMAX.28:= P2_Srobovanie.PAR.M4_AtlasCopcoInputs[3].4;
//    P2_Srobovanie.STAV.M4_Moment_ToleranciaMAX.29:= P2_Srobovanie.PAR.M4_AtlasCopcoInputs[3].5;
//    P2_Srobovanie.STAV.M4_Moment_ToleranciaMAX.30:= P2_Srobovanie.PAR.M4_AtlasCopcoInputs[3].6;
//    P2_Srobovanie.STAV.M4_Moment_ToleranciaMAX.31:= P2_Srobovanie.PAR.M4_AtlasCopcoInputs[3].7;
//    M4_Moment_ToleranciaMAX_REAL:= UDINT_TO_REAL(P2_Srobovanie.STAV.M4_Moment_ToleranciaMAX);
//    IF M4_Moment_ToleranciaMAX_REAL > 0 THEN
//        P2_Srobovanie.STAV.M4_Moment_ToleranciaMAX_REAL:= (M4_Moment_ToleranciaMAX_REAL*2.1)/131082;
//    ELSE
//        P2_Srobovanie.STAV.M4_Moment_ToleranciaMAX_REAL:= 0.0;
//    END_IF

    M4_PrevodMomentu.AtlasMaximalnaTolerancia:=P2_Srobovanie.PAR.M4_AtlasCopcoInputs[3];
    P2_Srobovanie.STAV.M4_Moment_ToleranciaMAX_REAL:=M4_PrevodMomentu.ToleranciaMAX;

    (*P2_Srobovanie.STAV.M4_Moment_ToleranciaMAX_REAL:= M4_Moment_ToleranciaMAX_REAL /100;*)

    //Moment - Tolerancia MIN//
//    P2_Srobovanie.STAV.M4_Moment_ToleranciaMIN.0:= P2_Srobovanie.PAR.M4_AtlasCopcoInputs[4].24;
//    P2_Srobovanie.STAV.M4_Moment_ToleranciaMIN.1:= P2_Srobovanie.PAR.M4_AtlasCopcoInputs[4].25;
//    P2_Srobovanie.STAV.M4_Moment_ToleranciaMIN.2:= P2_Srobovanie.PAR.M4_AtlasCopcoInputs[4].26;
//    P2_Srobovanie.STAV.M4_Moment_ToleranciaMIN.3:= P2_Srobovanie.PAR.M4_AtlasCopcoInputs[4].27;
//    P2_Srobovanie.STAV.M4_Moment_ToleranciaMIN.4:= P2_Srobovanie.PAR.M4_AtlasCopcoInputs[4].28;
//    P2_Srobovanie.STAV.M4_Moment_ToleranciaMIN.5:= P2_Srobovanie.PAR.M4_AtlasCopcoInputs[4].29;
//    P2_Srobovanie.STAV.M4_Moment_ToleranciaMIN.6:= P2_Srobovanie.PAR.M4_AtlasCopcoInputs[4].30;
//    P2_Srobovanie.STAV.M4_Moment_ToleranciaMIN.7:= P2_Srobovanie.PAR.M4_AtlasCopcoInputs[4].31;
//    P2_Srobovanie.STAV.M4_Moment_ToleranciaMIN.8:= P2_Srobovanie.PAR.M4_AtlasCopcoInputs[4].16;
//    P2_Srobovanie.STAV.M4_Moment_ToleranciaMIN.9:= P2_Srobovanie.PAR.M4_AtlasCopcoInputs[4].17;
//    P2_Srobovanie.STAV.M4_Moment_ToleranciaMIN.10:= P2_Srobovanie.PAR.M4_AtlasCopcoInputs[4].18;
//    P2_Srobovanie.STAV.M4_Moment_ToleranciaMIN.11:= P2_Srobovanie.PAR.M4_AtlasCopcoInputs[4].19;
//    P2_Srobovanie.STAV.M4_Moment_ToleranciaMIN.12:= P2_Srobovanie.PAR.M4_AtlasCopcoInputs[4].20;
//    P2_Srobovanie.STAV.M4_Moment_ToleranciaMIN.13:= P2_Srobovanie.PAR.M4_AtlasCopcoInputs[4].21;
//    P2_Srobovanie.STAV.M4_Moment_ToleranciaMIN.14:= P2_Srobovanie.PAR.M4_AtlasCopcoInputs[4].22;
//    P2_Srobovanie.STAV.M4_Moment_ToleranciaMIN.15:= P2_Srobovanie.PAR.M4_AtlasCopcoInputs[4].23;
//    P2_Srobovanie.STAV.M4_Moment_ToleranciaMIN.16:= P2_Srobovanie.PAR.M4_AtlasCopcoInputs[4].8;
//    P2_Srobovanie.STAV.M4_Moment_ToleranciaMIN.17:= P2_Srobovanie.PAR.M4_AtlasCopcoInputs[4].9;
//    P2_Srobovanie.STAV.M4_Moment_ToleranciaMIN.18:= P2_Srobovanie.PAR.M4_AtlasCopcoInputs[4].10;
//    P2_Srobovanie.STAV.M4_Moment_ToleranciaMIN.19:= P2_Srobovanie.PAR.M4_AtlasCopcoInputs[4].11;
//    P2_Srobovanie.STAV.M4_Moment_ToleranciaMIN.20:= P2_Srobovanie.PAR.M4_AtlasCopcoInputs[4].12;
//    P2_Srobovanie.STAV.M4_Moment_ToleranciaMIN.21:= P2_Srobovanie.PAR.M4_AtlasCopcoInputs[4].13;
//    P2_Srobovanie.STAV.M4_Moment_ToleranciaMIN.22:= P2_Srobovanie.PAR.M4_AtlasCopcoInputs[4].14;
//    P2_Srobovanie.STAV.M4_Moment_ToleranciaMIN.23:= P2_Srobovanie.PAR.M4_AtlasCopcoInputs[4].15;
//    P2_Srobovanie.STAV.M4_Moment_ToleranciaMIN.24:= P2_Srobovanie.PAR.M4_AtlasCopcoInputs[4].0;
//    P2_Srobovanie.STAV.M4_Moment_ToleranciaMIN.25:= P2_Srobovanie.PAR.M4_AtlasCopcoInputs[4].1;
//    P2_Srobovanie.STAV.M4_Moment_ToleranciaMIN.26:= P2_Srobovanie.PAR.M4_AtlasCopcoInputs[4].2;
//    P2_Srobovanie.STAV.M4_Moment_ToleranciaMIN.27:= P2_Srobovanie.PAR.M4_AtlasCopcoInputs[4].3;
//    P2_Srobovanie.STAV.M4_Moment_ToleranciaMIN.28:= P2_Srobovanie.PAR.M4_AtlasCopcoInputs[4].4;
//    P2_Srobovanie.STAV.M4_Moment_ToleranciaMIN.29:= P2_Srobovanie.PAR.M4_AtlasCopcoInputs[4].5;
//    P2_Srobovanie.STAV.M4_Moment_ToleranciaMIN.30:= P2_Srobovanie.PAR.M4_AtlasCopcoInputs[4].6;
//    P2_Srobovanie.STAV.M4_Moment_ToleranciaMIN.31:= P2_Srobovanie.PAR.M4_AtlasCopcoInputs[4].7;
//    M4_Moment_ToleranciaMIN_REAL:= UDINT_TO_REAL(P2_Srobovanie.STAV.M4_Moment_ToleranciaMIN);
//    IF M4_Moment_ToleranciaMIN_REAL > 0 THEN
//        P2_Srobovanie.STAV.M4_Moment_ToleranciaMIN_REAL:= (M4_Moment_ToleranciaMIN_REAL*2.1)/131082;
//    ELSE
//        P2_Srobovanie.STAV.M4_Moment_ToleranciaMIN_REAL:= 0.0;
//    END_IF
//

    M4_PrevodMomentu.AtlasMinimalnaTolerancia:=P2_Srobovanie.PAR.M4_AtlasCopcoInputs[4];
    P2_Srobovanie.STAV.M4_Moment_ToleranciaMIN_REAL:=M4_PrevodMomentu.ToleranciaMIN;

    (*P2_Srobovanie.STAV.M4_Moment_ToleranciaMIN_REAL:= M4_Moment_ToleranciaMIN_REAL /100;*)

    //Dosiahnutý úhol//
    P2_Srobovanie.STAV.M4_DosiahnutyUhol.0:= P2_Srobovanie.PAR.M4_AtlasCopcoInputs[0].24;
    P2_Srobovanie.STAV.M4_DosiahnutyUhol.1:= P2_Srobovanie.PAR.M4_AtlasCopcoInputs[0].25;
    P2_Srobovanie.STAV.M4_DosiahnutyUhol.2:= P2_Srobovanie.PAR.M4_AtlasCopcoInputs[0].26;
    P2_Srobovanie.STAV.M4_DosiahnutyUhol.3:= P2_Srobovanie.PAR.M4_AtlasCopcoInputs[0].27;
    P2_Srobovanie.STAV.M4_DosiahnutyUhol.4:= P2_Srobovanie.PAR.M4_AtlasCopcoInputs[0].28;
    P2_Srobovanie.STAV.M4_DosiahnutyUhol.5:= P2_Srobovanie.PAR.M4_AtlasCopcoInputs[0].29;
    P2_Srobovanie.STAV.M4_DosiahnutyUhol.6:= P2_Srobovanie.PAR.M4_AtlasCopcoInputs[0].30;
    P2_Srobovanie.STAV.M4_DosiahnutyUhol.7:= P2_Srobovanie.PAR.M4_AtlasCopcoInputs[0].31;
    P2_Srobovanie.STAV.M4_DosiahnutyUhol.8:= P2_Srobovanie.PAR.M4_AtlasCopcoInputs[0].16;
    P2_Srobovanie.STAV.M4_DosiahnutyUhol.9:= P2_Srobovanie.PAR.M4_AtlasCopcoInputs[0].17;
    P2_Srobovanie.STAV.M4_DosiahnutyUhol.10:= P2_Srobovanie.PAR.M4_AtlasCopcoInputs[0].18;
    P2_Srobovanie.STAV.M4_DosiahnutyUhol.11:= P2_Srobovanie.PAR.M4_AtlasCopcoInputs[0].19;
    P2_Srobovanie.STAV.M4_DosiahnutyUhol.12:= P2_Srobovanie.PAR.M4_AtlasCopcoInputs[0].20;
    P2_Srobovanie.STAV.M4_DosiahnutyUhol.13:= P2_Srobovanie.PAR.M4_AtlasCopcoInputs[0].21;
    P2_Srobovanie.STAV.M4_DosiahnutyUhol.14:= P2_Srobovanie.PAR.M4_AtlasCopcoInputs[0].22;
    P2_Srobovanie.STAV.M4_DosiahnutyUhol.15:= P2_Srobovanie.PAR.M4_AtlasCopcoInputs[0].23;

    //Uhol - Tolerancia MAX//
    P2_Srobovanie.STAV.M4_Uhol_ToleranciaMAX.0:= P2_Srobovanie.PAR.M4_AtlasCopcoInputs[2].8;
    P2_Srobovanie.STAV.M4_Uhol_ToleranciaMAX.1:= P2_Srobovanie.PAR.M4_AtlasCopcoInputs[2].9;
    P2_Srobovanie.STAV.M4_Uhol_ToleranciaMAX.2:= P2_Srobovanie.PAR.M4_AtlasCopcoInputs[2].10;
    P2_Srobovanie.STAV.M4_Uhol_ToleranciaMAX.3:= P2_Srobovanie.PAR.M4_AtlasCopcoInputs[2].11;
    P2_Srobovanie.STAV.M4_Uhol_ToleranciaMAX.4:= P2_Srobovanie.PAR.M4_AtlasCopcoInputs[2].12;
    P2_Srobovanie.STAV.M4_Uhol_ToleranciaMAX.5:= P2_Srobovanie.PAR.M4_AtlasCopcoInputs[2].13;
    P2_Srobovanie.STAV.M4_Uhol_ToleranciaMAX.6:= P2_Srobovanie.PAR.M4_AtlasCopcoInputs[2].14;
    P2_Srobovanie.STAV.M4_Uhol_ToleranciaMAX.7:= P2_Srobovanie.PAR.M4_AtlasCopcoInputs[2].15;
    P2_Srobovanie.STAV.M4_Uhol_ToleranciaMAX.8:= P2_Srobovanie.PAR.M4_AtlasCopcoInputs[2].0;
    P2_Srobovanie.STAV.M4_Uhol_ToleranciaMAX.9:= P2_Srobovanie.PAR.M4_AtlasCopcoInputs[2].1;
    P2_Srobovanie.STAV.M4_Uhol_ToleranciaMAX.10:= P2_Srobovanie.PAR.M4_AtlasCopcoInputs[2].2;
    P2_Srobovanie.STAV.M4_Uhol_ToleranciaMAX.11:= P2_Srobovanie.PAR.M4_AtlasCopcoInputs[2].3;
    P2_Srobovanie.STAV.M4_Uhol_ToleranciaMAX.12:= P2_Srobovanie.PAR.M4_AtlasCopcoInputs[2].4;
    P2_Srobovanie.STAV.M4_Uhol_ToleranciaMAX.13:= P2_Srobovanie.PAR.M4_AtlasCopcoInputs[2].5;
    P2_Srobovanie.STAV.M4_Uhol_ToleranciaMAX.14:= P2_Srobovanie.PAR.M4_AtlasCopcoInputs[2].6;
    P2_Srobovanie.STAV.M4_Uhol_ToleranciaMAX.15:= P2_Srobovanie.PAR.M4_AtlasCopcoInputs[2].7;

    //Uhol - Tolerancia MIN//
    P2_Srobovanie.STAV.M4_Uhol_ToleranciaMIN.0:= P2_Srobovanie.PAR.M4_AtlasCopcoInputs[2].24;
    P2_Srobovanie.STAV.M4_Uhol_ToleranciaMIN.1:= P2_Srobovanie.PAR.M4_AtlasCopcoInputs[2].25;
    P2_Srobovanie.STAV.M4_Uhol_ToleranciaMIN.2:= P2_Srobovanie.PAR.M4_AtlasCopcoInputs[2].26;
    P2_Srobovanie.STAV.M4_Uhol_ToleranciaMIN.3:= P2_Srobovanie.PAR.M4_AtlasCopcoInputs[2].27;
    P2_Srobovanie.STAV.M4_Uhol_ToleranciaMIN.4:= P2_Srobovanie.PAR.M4_AtlasCopcoInputs[2].28;
    P2_Srobovanie.STAV.M4_Uhol_ToleranciaMIN.5:= P2_Srobovanie.PAR.M4_AtlasCopcoInputs[2].29;
    P2_Srobovanie.STAV.M4_Uhol_ToleranciaMIN.6:= P2_Srobovanie.PAR.M4_AtlasCopcoInputs[2].30;
    P2_Srobovanie.STAV.M4_Uhol_ToleranciaMIN.7:= P2_Srobovanie.PAR.M4_AtlasCopcoInputs[2].31;
    P2_Srobovanie.STAV.M4_Uhol_ToleranciaMIN.8:= P2_Srobovanie.PAR.M4_AtlasCopcoInputs[2].16;
    P2_Srobovanie.STAV.M4_Uhol_ToleranciaMIN.9:= P2_Srobovanie.PAR.M4_AtlasCopcoInputs[2].17;
    P2_Srobovanie.STAV.M4_Uhol_ToleranciaMIN.10:= P2_Srobovanie.PAR.M4_AtlasCopcoInputs[2].18;
    P2_Srobovanie.STAV.M4_Uhol_ToleranciaMIN.11:= P2_Srobovanie.PAR.M4_AtlasCopcoInputs[2].19;
    P2_Srobovanie.STAV.M4_Uhol_ToleranciaMIN.12:= P2_Srobovanie.PAR.M4_AtlasCopcoInputs[2].20;
    P2_Srobovanie.STAV.M4_Uhol_ToleranciaMIN.13:= P2_Srobovanie.PAR.M4_AtlasCopcoInputs[2].21;
    P2_Srobovanie.STAV.M4_Uhol_ToleranciaMIN.14:= P2_Srobovanie.PAR.M4_AtlasCopcoInputs[2].22;
    P2_Srobovanie.STAV.M4_Uhol_ToleranciaMIN.15:= P2_Srobovanie.PAR.M4_AtlasCopcoInputs[2].23;

    //*************************************************************Skrutkovacka M6*******************************************************************************//
    //Vstupy z AtlasCopco do PLC//
    P2_Srobovanie.Skrutkovacka_M6.Stav_VysledokPotvrdeny:= P2_Srobovanie.PAR.M6_AtlasCopcoInputs[0].0;
    P2_Srobovanie.Skrutkovacka_M6.Stav_EmergencyStop:= P2_Srobovanie.PAR.M6_AtlasCopcoInputs[0].1;
    P2_Srobovanie.Skrutkovacka_M6.Stav_READY_to_START:= P2_Srobovanie.PAR.M6_AtlasCopcoInputs[0].2;
    P2_Srobovanie.Skrutkovacka_M6.Stav_MANUAL:= P2_Srobovanie.PAR.M6_AtlasCopcoInputs[0].3;
    P2_Srobovanie.Skrutkovacka_M6.Stav_UtahovanieUkoncene:= P2_Srobovanie.PAR.M6_AtlasCopcoInputs[0].4;
    P2_Srobovanie.Skrutkovacka_M6.Stav_VysledokUtahovania_NG:= P2_Srobovanie.PAR.M6_AtlasCopcoInputs[0].5;
    P2_Srobovanie.Skrutkovacka_M6.Stav_VysledokUtahovania_OK:= P2_Srobovanie.PAR.M6_AtlasCopcoInputs[0].6;
    P2_Srobovanie.Skrutkovacka_M6.Stav_SmerOtacania_VPRED:= P2_Srobovanie.PAR.M6_AtlasCopcoInputs[0].7;
    P2_Srobovanie.Skrutkovacka_M6.Stav_BUSY:= P2_Srobovanie.PAR.M6_AtlasCopcoInputs[0].8;
    P2_Srobovanie.Skrutkovacka_M6.Stav_ControlerSwitch_ON:= P2_Srobovanie.PAR.M6_AtlasCopcoInputs[0].9;
    P2_Srobovanie.Skrutkovacka_M6.Stav_Station_READY:= P2_Srobovanie.PAR.M6_AtlasCopcoInputs[0].10;
    P2_Srobovanie.Skrutkovacka_M6.Stav_NastrojPripojeny:= P2_Srobovanie.PAR.M6_AtlasCopcoInputs[0].11;
    P2_Srobovanie.Skrutkovacka_M6.Stav_NastrojUtahuje:= P2_Srobovanie.PAR.M6_AtlasCopcoInputs[0].12;

    //Výstupy z PLC do AtlasCopco//
    P2_Srobovanie.PAR.M6_AllasCopcoOutputs[0].0:= P2_Srobovanie.Skrutkovacka_M6.RESET_Poruchy;
    P2_Srobovanie.PAR.M6_AllasCopcoOutputs[0].1:= P2_Srobovanie.Skrutkovacka_M6.RESET_Vysledkov;
    P2_Srobovanie.PAR.M6_AllasCopcoOutputs[0].2:= P2_Srobovanie.Skrutkovacka_M6.START_Skrutkovania;
    P2_Srobovanie.PAR.M6_AllasCopcoOutputs[0].3:= P2_Srobovanie.Skrutkovacka_M6.START_Utahovania;

    //Dosiahnutý moment//
//    P2_Srobovanie.STAV.M6_DosiahnutyMoment.0:= P2_Srobovanie.PAR.M6_AtlasCopcoInputs[1].24;
//    P2_Srobovanie.STAV.M6_DosiahnutyMoment.1:= P2_Srobovanie.PAR.M6_AtlasCopcoInputs[1].25;
//    P2_Srobovanie.STAV.M6_DosiahnutyMoment.2:= P2_Srobovanie.PAR.M6_AtlasCopcoInputs[1].26;
//    P2_Srobovanie.STAV.M6_DosiahnutyMoment.3:= P2_Srobovanie.PAR.M6_AtlasCopcoInputs[1].27;
//    P2_Srobovanie.STAV.M6_DosiahnutyMoment.4:= P2_Srobovanie.PAR.M6_AtlasCopcoInputs[1].28;
//    P2_Srobovanie.STAV.M6_DosiahnutyMoment.5:= P2_Srobovanie.PAR.M6_AtlasCopcoInputs[1].29;
//    P2_Srobovanie.STAV.M6_DosiahnutyMoment.6:= P2_Srobovanie.PAR.M6_AtlasCopcoInputs[1].30;
//    P2_Srobovanie.STAV.M6_DosiahnutyMoment.7:= P2_Srobovanie.PAR.M6_AtlasCopcoInputs[1].31;
//    P2_Srobovanie.STAV.M6_DosiahnutyMoment.8:= P2_Srobovanie.PAR.M6_AtlasCopcoInputs[1].16;
//    P2_Srobovanie.STAV.M6_DosiahnutyMoment.9:= P2_Srobovanie.PAR.M6_AtlasCopcoInputs[1].17;
//    P2_Srobovanie.STAV.M6_DosiahnutyMoment.10:= P2_Srobovanie.PAR.M6_AtlasCopcoInputs[1].18;
//    P2_Srobovanie.STAV.M6_DosiahnutyMoment.11:= P2_Srobovanie.PAR.M6_AtlasCopcoInputs[1].19;
//    P2_Srobovanie.STAV.M6_DosiahnutyMoment.12:= P2_Srobovanie.PAR.M6_AtlasCopcoInputs[1].20;
//    P2_Srobovanie.STAV.M6_DosiahnutyMoment.13:= P2_Srobovanie.PAR.M6_AtlasCopcoInputs[1].21;
//    P2_Srobovanie.STAV.M6_DosiahnutyMoment.14:= P2_Srobovanie.PAR.M6_AtlasCopcoInputs[1].22;
//    P2_Srobovanie.STAV.M6_DosiahnutyMoment.15:= P2_Srobovanie.PAR.M6_AtlasCopcoInputs[1].23;
//    P2_Srobovanie.STAV.M6_DosiahnutyMoment.16:= P2_Srobovanie.PAR.M6_AtlasCopcoInputs[1].8;
//    P2_Srobovanie.STAV.M6_DosiahnutyMoment.17:= P2_Srobovanie.PAR.M6_AtlasCopcoInputs[1].9;
//    P2_Srobovanie.STAV.M6_DosiahnutyMoment.18:= P2_Srobovanie.PAR.M6_AtlasCopcoInputs[1].10;
//    P2_Srobovanie.STAV.M6_DosiahnutyMoment.19:= P2_Srobovanie.PAR.M6_AtlasCopcoInputs[1].11;
//    P2_Srobovanie.STAV.M6_DosiahnutyMoment.20:= P2_Srobovanie.PAR.M6_AtlasCopcoInputs[1].12;
//    P2_Srobovanie.STAV.M6_DosiahnutyMoment.21:= P2_Srobovanie.PAR.M6_AtlasCopcoInputs[1].13;
//    P2_Srobovanie.STAV.M6_DosiahnutyMoment.22:= P2_Srobovanie.PAR.M6_AtlasCopcoInputs[1].14;
//    P2_Srobovanie.STAV.M6_DosiahnutyMoment.23:= P2_Srobovanie.PAR.M6_AtlasCopcoInputs[1].15;
//    P2_Srobovanie.STAV.M6_DosiahnutyMoment.24:= P2_Srobovanie.PAR.M6_AtlasCopcoInputs[1].0;
//    P2_Srobovanie.STAV.M6_DosiahnutyMoment.25:= P2_Srobovanie.PAR.M6_AtlasCopcoInputs[1].1;
//    P2_Srobovanie.STAV.M6_DosiahnutyMoment.26:= P2_Srobovanie.PAR.M6_AtlasCopcoInputs[1].2;
//    P2_Srobovanie.STAV.M6_DosiahnutyMoment.27:= P2_Srobovanie.PAR.M6_AtlasCopcoInputs[1].3;
//    P2_Srobovanie.STAV.M6_DosiahnutyMoment.28:= P2_Srobovanie.PAR.M6_AtlasCopcoInputs[1].4;
//    P2_Srobovanie.STAV.M6_DosiahnutyMoment.29:= P2_Srobovanie.PAR.M6_AtlasCopcoInputs[1].5;
//    P2_Srobovanie.STAV.M6_DosiahnutyMoment.30:= P2_Srobovanie.PAR.M6_AtlasCopcoInputs[1].6;
//    P2_Srobovanie.STAV.M6_DosiahnutyMoment.31:= P2_Srobovanie.PAR.M6_AtlasCopcoInputs[1].7;
//    M6_DosiahnutyMoment_REAL:= UDINT_TO_REAL(P2_Srobovanie.STAV.M6_DosiahnutyMoment);
//    IF M6_DosiahnutyMoment_REAL > 0 THEN
//       P2_Srobovanie.STAV.M6_DosiahnutyMoment_REAL:= (M6_DosiahnutyMoment_REAL*7.2)/458772;
//    ELSE
//        P2_Srobovanie.STAV.M6_DosiahnutyMoment_REAL:= 0.0;
//    END_IF

    M6_PrevodMomentu.AtlasAktualnyMoment:=P2_Srobovanie.PAR.M6_AtlasCopcoInputs[1];
    P2_Srobovanie.STAV.M6_DosiahnutyMoment_REAL:=M6_PrevodMomentu.AktualnyMoment;

    (*P2_Srobovanie.STAV.M6_DosiahnutyMoment_REAL:= M6_DosiahnutyMoment_REAL /100;*)

    //Moment - Tolerancia MAX//
//    P2_Srobovanie.STAV.M6_Moment_ToleranciaMAX.0:= P2_Srobovanie.PAR.M6_AtlasCopcoInputs[3].24;
//    P2_Srobovanie.STAV.M6_Moment_ToleranciaMAX.1:= P2_Srobovanie.PAR.M6_AtlasCopcoInputs[3].25;
//    P2_Srobovanie.STAV.M6_Moment_ToleranciaMAX.2:= P2_Srobovanie.PAR.M6_AtlasCopcoInputs[3].26;
//    P2_Srobovanie.STAV.M6_Moment_ToleranciaMAX.3:= P2_Srobovanie.PAR.M6_AtlasCopcoInputs[3].27;
//    P2_Srobovanie.STAV.M6_Moment_ToleranciaMAX.4:= P2_Srobovanie.PAR.M6_AtlasCopcoInputs[3].28;
//    P2_Srobovanie.STAV.M6_Moment_ToleranciaMAX.5:= P2_Srobovanie.PAR.M6_AtlasCopcoInputs[3].29;
//    P2_Srobovanie.STAV.M6_Moment_ToleranciaMAX.6:= P2_Srobovanie.PAR.M6_AtlasCopcoInputs[3].30;
//    P2_Srobovanie.STAV.M6_Moment_ToleranciaMAX.7:= P2_Srobovanie.PAR.M6_AtlasCopcoInputs[3].31;
//    P2_Srobovanie.STAV.M6_Moment_ToleranciaMAX.8:= P2_Srobovanie.PAR.M6_AtlasCopcoInputs[3].16;
//    P2_Srobovanie.STAV.M6_Moment_ToleranciaMAX.9:= P2_Srobovanie.PAR.M6_AtlasCopcoInputs[3].17;
//    P2_Srobovanie.STAV.M6_Moment_ToleranciaMAX.10:= P2_Srobovanie.PAR.M6_AtlasCopcoInputs[3].18;
//    P2_Srobovanie.STAV.M6_Moment_ToleranciaMAX.11:= P2_Srobovanie.PAR.M6_AtlasCopcoInputs[3].19;
//    P2_Srobovanie.STAV.M6_Moment_ToleranciaMAX.12:= P2_Srobovanie.PAR.M6_AtlasCopcoInputs[3].20;
//    P2_Srobovanie.STAV.M6_Moment_ToleranciaMAX.13:= P2_Srobovanie.PAR.M6_AtlasCopcoInputs[3].21;
//    P2_Srobovanie.STAV.M6_Moment_ToleranciaMAX.14:= P2_Srobovanie.PAR.M6_AtlasCopcoInputs[3].22;
//    P2_Srobovanie.STAV.M6_Moment_ToleranciaMAX.15:= P2_Srobovanie.PAR.M6_AtlasCopcoInputs[3].23;
//    P2_Srobovanie.STAV.M6_Moment_ToleranciaMAX.16:= P2_Srobovanie.PAR.M6_AtlasCopcoInputs[3].8;
//    P2_Srobovanie.STAV.M6_Moment_ToleranciaMAX.17:= P2_Srobovanie.PAR.M6_AtlasCopcoInputs[3].9;
//    P2_Srobovanie.STAV.M6_Moment_ToleranciaMAX.18:= P2_Srobovanie.PAR.M6_AtlasCopcoInputs[3].10;
//    P2_Srobovanie.STAV.M6_Moment_ToleranciaMAX.19:= P2_Srobovanie.PAR.M6_AtlasCopcoInputs[3].11;
//    P2_Srobovanie.STAV.M6_Moment_ToleranciaMAX.20:= P2_Srobovanie.PAR.M6_AtlasCopcoInputs[3].12;
//    P2_Srobovanie.STAV.M6_Moment_ToleranciaMAX.21:= P2_Srobovanie.PAR.M6_AtlasCopcoInputs[3].13;
//    P2_Srobovanie.STAV.M6_Moment_ToleranciaMAX.22:= P2_Srobovanie.PAR.M6_AtlasCopcoInputs[3].14;
//    P2_Srobovanie.STAV.M6_Moment_ToleranciaMAX.23:= P2_Srobovanie.PAR.M6_AtlasCopcoInputs[3].15;
//    P2_Srobovanie.STAV.M6_Moment_ToleranciaMAX.24:= P2_Srobovanie.PAR.M6_AtlasCopcoInputs[3].0;
//    P2_Srobovanie.STAV.M6_Moment_ToleranciaMAX.25:= P2_Srobovanie.PAR.M6_AtlasCopcoInputs[3].1;
//    P2_Srobovanie.STAV.M6_Moment_ToleranciaMAX.26:= P2_Srobovanie.PAR.M6_AtlasCopcoInputs[3].2;
//    P2_Srobovanie.STAV.M6_Moment_ToleranciaMAX.27:= P2_Srobovanie.PAR.M6_AtlasCopcoInputs[3].3;
//    P2_Srobovanie.STAV.M6_Moment_ToleranciaMAX.28:= P2_Srobovanie.PAR.M6_AtlasCopcoInputs[3].4;
//    P2_Srobovanie.STAV.M6_Moment_ToleranciaMAX.29:= P2_Srobovanie.PAR.M6_AtlasCopcoInputs[3].5;
//    P2_Srobovanie.STAV.M6_Moment_ToleranciaMAX.30:= P2_Srobovanie.PAR.M6_AtlasCopcoInputs[3].6;
//    P2_Srobovanie.STAV.M6_Moment_ToleranciaMAX.31:= P2_Srobovanie.PAR.M6_AtlasCopcoInputs[3].7;
//    M6_Moment_ToleranciaMAX_REAL:= UDINT_TO_REAL(P2_Srobovanie.STAV.M6_Moment_ToleranciaMAX);
//    IF M6_Moment_ToleranciaMAX_REAL > 0 THEN
//        P2_Srobovanie.STAV.M6_Moment_ToleranciaMAX_REAL:= (M6_Moment_ToleranciaMAX_REAL*7.2)/458772;
//    ELSE
//        P2_Srobovanie.STAV.M6_Moment_ToleranciaMAX_REAL:= 0.0;
//    END_IF
//

    M6_PrevodMomentu.AtlasMaximalnaTolerancia:=P2_Srobovanie.PAR.M6_AtlasCopcoInputs[3];
    P2_Srobovanie.STAV.M6_Moment_ToleranciaMAX_REAL:=M6_PrevodMomentu.ToleranciaMAX;

    (*P2_Srobovanie.STAV.M6_Moment_ToleranciaMAX_REAL:= M6_Moment_ToleranciaMAX_REAL /100;*)

    //Moment - Tolerancia MIN//
//    P2_Srobovanie.STAV.M6_Moment_ToleranciaMIN.0:= P2_Srobovanie.PAR.M6_AtlasCopcoInputs[4].24;
//    P2_Srobovanie.STAV.M6_Moment_ToleranciaMIN.1:= P2_Srobovanie.PAR.M6_AtlasCopcoInputs[4].25;
//    P2_Srobovanie.STAV.M6_Moment_ToleranciaMIN.2:= P2_Srobovanie.PAR.M6_AtlasCopcoInputs[4].26;
//    P2_Srobovanie.STAV.M6_Moment_ToleranciaMIN.3:= P2_Srobovanie.PAR.M6_AtlasCopcoInputs[4].27;
//    P2_Srobovanie.STAV.M6_Moment_ToleranciaMIN.4:= P2_Srobovanie.PAR.M6_AtlasCopcoInputs[4].28;
//    P2_Srobovanie.STAV.M6_Moment_ToleranciaMIN.5:= P2_Srobovanie.PAR.M6_AtlasCopcoInputs[4].29;
//    P2_Srobovanie.STAV.M6_Moment_ToleranciaMIN.6:= P2_Srobovanie.PAR.M6_AtlasCopcoInputs[4].30;
//    P2_Srobovanie.STAV.M6_Moment_ToleranciaMIN.7:= P2_Srobovanie.PAR.M6_AtlasCopcoInputs[4].31;
//    P2_Srobovanie.STAV.M6_Moment_ToleranciaMIN.8:= P2_Srobovanie.PAR.M6_AtlasCopcoInputs[4].16;
//    P2_Srobovanie.STAV.M6_Moment_ToleranciaMIN.9:= P2_Srobovanie.PAR.M6_AtlasCopcoInputs[4].17;
//    P2_Srobovanie.STAV.M6_Moment_ToleranciaMIN.10:= P2_Srobovanie.PAR.M6_AtlasCopcoInputs[4].18;
//    P2_Srobovanie.STAV.M6_Moment_ToleranciaMIN.11:= P2_Srobovanie.PAR.M6_AtlasCopcoInputs[4].19;
//    P2_Srobovanie.STAV.M6_Moment_ToleranciaMIN.12:= P2_Srobovanie.PAR.M6_AtlasCopcoInputs[4].20;
//    P2_Srobovanie.STAV.M6_Moment_ToleranciaMIN.13:= P2_Srobovanie.PAR.M6_AtlasCopcoInputs[4].21;
//    P2_Srobovanie.STAV.M6_Moment_ToleranciaMIN.14:= P2_Srobovanie.PAR.M6_AtlasCopcoInputs[4].22;
//    P2_Srobovanie.STAV.M6_Moment_ToleranciaMIN.15:= P2_Srobovanie.PAR.M6_AtlasCopcoInputs[4].23;
//    P2_Srobovanie.STAV.M6_Moment_ToleranciaMIN.16:= P2_Srobovanie.PAR.M6_AtlasCopcoInputs[4].8;
//    P2_Srobovanie.STAV.M6_Moment_ToleranciaMIN.17:= P2_Srobovanie.PAR.M6_AtlasCopcoInputs[4].9;
//    P2_Srobovanie.STAV.M6_Moment_ToleranciaMIN.18:= P2_Srobovanie.PAR.M6_AtlasCopcoInputs[4].10;
//    P2_Srobovanie.STAV.M6_Moment_ToleranciaMIN.19:= P2_Srobovanie.PAR.M6_AtlasCopcoInputs[4].11;
//    P2_Srobovanie.STAV.M6_Moment_ToleranciaMIN.20:= P2_Srobovanie.PAR.M6_AtlasCopcoInputs[4].12;
//    P2_Srobovanie.STAV.M6_Moment_ToleranciaMIN.21:= P2_Srobovanie.PAR.M6_AtlasCopcoInputs[4].13;
//    P2_Srobovanie.STAV.M6_Moment_ToleranciaMIN.22:= P2_Srobovanie.PAR.M6_AtlasCopcoInputs[4].14;
//    P2_Srobovanie.STAV.M6_Moment_ToleranciaMIN.23:= P2_Srobovanie.PAR.M6_AtlasCopcoInputs[4].15;
//    P2_Srobovanie.STAV.M6_Moment_ToleranciaMIN.24:= P2_Srobovanie.PAR.M6_AtlasCopcoInputs[4].0;
//    P2_Srobovanie.STAV.M6_Moment_ToleranciaMIN.25:= P2_Srobovanie.PAR.M6_AtlasCopcoInputs[4].1;
//    P2_Srobovanie.STAV.M6_Moment_ToleranciaMIN.26:= P2_Srobovanie.PAR.M6_AtlasCopcoInputs[4].2;
//    P2_Srobovanie.STAV.M6_Moment_ToleranciaMIN.27:= P2_Srobovanie.PAR.M6_AtlasCopcoInputs[4].3;
//    P2_Srobovanie.STAV.M6_Moment_ToleranciaMIN.28:= P2_Srobovanie.PAR.M6_AtlasCopcoInputs[4].4;
//    P2_Srobovanie.STAV.M6_Moment_ToleranciaMIN.29:= P2_Srobovanie.PAR.M6_AtlasCopcoInputs[4].5;
//    P2_Srobovanie.STAV.M6_Moment_ToleranciaMIN.30:= P2_Srobovanie.PAR.M6_AtlasCopcoInputs[4].6;
//    P2_Srobovanie.STAV.M6_Moment_ToleranciaMIN.31:= P2_Srobovanie.PAR.M6_AtlasCopcoInputs[4].7;
//    M6_Moment_ToleranciaMIN_REAL:= UDINT_TO_REAL(P2_Srobovanie.STAV.M6_Moment_ToleranciaMIN);
//    IF M6_Moment_ToleranciaMIN_REAL > 0 THEN
//        P2_Srobovanie.STAV.M6_Moment_ToleranciaMIN_REAL:= (M6_Moment_ToleranciaMIN_REAL*7.2)/458772;
//    ELSE
//        P2_Srobovanie.STAV.M6_Moment_ToleranciaMIN_REAL:= 0.0;
//    END_IF

    M6_PrevodMomentu.AtlasMinimalnaTolerancia:=P2_Srobovanie.PAR.M6_AtlasCopcoInputs[4];
    P2_Srobovanie.STAV.M6_Moment_ToleranciaMIN_REAL:=M6_PrevodMomentu.ToleranciaMIN;

    (*P2_Srobovanie.STAV.M6_Moment_ToleranciaMIN_REAL:= M6_Moment_ToleranciaMIN_REAL /100;*)

    //Dosiahnutý úhol//
    P2_Srobovanie.STAV.M6_DosiahnutyUhol.0:= P2_Srobovanie.PAR.M6_AtlasCopcoInputs[0].24;
    P2_Srobovanie.STAV.M6_DosiahnutyUhol.1:= P2_Srobovanie.PAR.M6_AtlasCopcoInputs[0].25;
    P2_Srobovanie.STAV.M6_DosiahnutyUhol.2:= P2_Srobovanie.PAR.M6_AtlasCopcoInputs[0].26;
    P2_Srobovanie.STAV.M6_DosiahnutyUhol.3:= P2_Srobovanie.PAR.M6_AtlasCopcoInputs[0].27;
    P2_Srobovanie.STAV.M6_DosiahnutyUhol.4:= P2_Srobovanie.PAR.M6_AtlasCopcoInputs[0].28;
    P2_Srobovanie.STAV.M6_DosiahnutyUhol.5:= P2_Srobovanie.PAR.M6_AtlasCopcoInputs[0].29;
    P2_Srobovanie.STAV.M6_DosiahnutyUhol.6:= P2_Srobovanie.PAR.M6_AtlasCopcoInputs[0].30;
    P2_Srobovanie.STAV.M6_DosiahnutyUhol.7:= P2_Srobovanie.PAR.M6_AtlasCopcoInputs[0].31;
    P2_Srobovanie.STAV.M6_DosiahnutyUhol.8:= P2_Srobovanie.PAR.M6_AtlasCopcoInputs[0].16;
    P2_Srobovanie.STAV.M6_DosiahnutyUhol.9:= P2_Srobovanie.PAR.M6_AtlasCopcoInputs[0].17;
    P2_Srobovanie.STAV.M6_DosiahnutyUhol.10:= P2_Srobovanie.PAR.M6_AtlasCopcoInputs[0].18;
    P2_Srobovanie.STAV.M6_DosiahnutyUhol.11:= P2_Srobovanie.PAR.M6_AtlasCopcoInputs[0].19;
    P2_Srobovanie.STAV.M6_DosiahnutyUhol.12:= P2_Srobovanie.PAR.M6_AtlasCopcoInputs[0].20;
    P2_Srobovanie.STAV.M6_DosiahnutyUhol.13:= P2_Srobovanie.PAR.M6_AtlasCopcoInputs[0].21;
    P2_Srobovanie.STAV.M6_DosiahnutyUhol.14:= P2_Srobovanie.PAR.M6_AtlasCopcoInputs[0].22;
    P2_Srobovanie.STAV.M6_DosiahnutyUhol.15:= P2_Srobovanie.PAR.M6_AtlasCopcoInputs[0].23;

    //Uhol - Tolerancia MAX//
    P2_Srobovanie.STAV.M6_Uhol_ToleranciaMAX.0:= P2_Srobovanie.PAR.M6_AtlasCopcoInputs[2].8;
    P2_Srobovanie.STAV.M6_Uhol_ToleranciaMAX.1:= P2_Srobovanie.PAR.M6_AtlasCopcoInputs[2].9;
    P2_Srobovanie.STAV.M6_Uhol_ToleranciaMAX.2:= P2_Srobovanie.PAR.M6_AtlasCopcoInputs[2].10;
    P2_Srobovanie.STAV.M6_Uhol_ToleranciaMAX.3:= P2_Srobovanie.PAR.M6_AtlasCopcoInputs[2].11;
    P2_Srobovanie.STAV.M6_Uhol_ToleranciaMAX.4:= P2_Srobovanie.PAR.M6_AtlasCopcoInputs[2].12;
    P2_Srobovanie.STAV.M6_Uhol_ToleranciaMAX.5:= P2_Srobovanie.PAR.M6_AtlasCopcoInputs[2].13;
    P2_Srobovanie.STAV.M6_Uhol_ToleranciaMAX.6:= P2_Srobovanie.PAR.M6_AtlasCopcoInputs[2].14;
    P2_Srobovanie.STAV.M6_Uhol_ToleranciaMAX.7:= P2_Srobovanie.PAR.M6_AtlasCopcoInputs[2].15;
    P2_Srobovanie.STAV.M6_Uhol_ToleranciaMAX.8:= P2_Srobovanie.PAR.M6_AtlasCopcoInputs[2].0;
    P2_Srobovanie.STAV.M6_Uhol_ToleranciaMAX.9:= P2_Srobovanie.PAR.M6_AtlasCopcoInputs[2].1;
    P2_Srobovanie.STAV.M6_Uhol_ToleranciaMAX.10:= P2_Srobovanie.PAR.M6_AtlasCopcoInputs[2].2;
    P2_Srobovanie.STAV.M6_Uhol_ToleranciaMAX.11:= P2_Srobovanie.PAR.M6_AtlasCopcoInputs[2].3;
    P2_Srobovanie.STAV.M6_Uhol_ToleranciaMAX.12:= P2_Srobovanie.PAR.M6_AtlasCopcoInputs[2].4;
    P2_Srobovanie.STAV.M6_Uhol_ToleranciaMAX.13:= P2_Srobovanie.PAR.M6_AtlasCopcoInputs[2].5;
    P2_Srobovanie.STAV.M6_Uhol_ToleranciaMAX.14:= P2_Srobovanie.PAR.M6_AtlasCopcoInputs[2].6;
    P2_Srobovanie.STAV.M6_Uhol_ToleranciaMAX.15:= P2_Srobovanie.PAR.M6_AtlasCopcoInputs[2].7;

    //Uhol - Tolerancia MIN//
    P2_Srobovanie.STAV.M6_Uhol_ToleranciaMIN.0:= P2_Srobovanie.PAR.M6_AtlasCopcoInputs[2].24;
    P2_Srobovanie.STAV.M6_Uhol_ToleranciaMIN.1:= P2_Srobovanie.PAR.M6_AtlasCopcoInputs[2].25;
    P2_Srobovanie.STAV.M6_Uhol_ToleranciaMIN.2:= P2_Srobovanie.PAR.M6_AtlasCopcoInputs[2].26;
    P2_Srobovanie.STAV.M6_Uhol_ToleranciaMIN.3:= P2_Srobovanie.PAR.M6_AtlasCopcoInputs[2].27;
    P2_Srobovanie.STAV.M6_Uhol_ToleranciaMIN.4:= P2_Srobovanie.PAR.M6_AtlasCopcoInputs[2].28;
    P2_Srobovanie.STAV.M6_Uhol_ToleranciaMIN.5:= P2_Srobovanie.PAR.M6_AtlasCopcoInputs[2].29;
    P2_Srobovanie.STAV.M6_Uhol_ToleranciaMIN.6:= P2_Srobovanie.PAR.M6_AtlasCopcoInputs[2].30;
    P2_Srobovanie.STAV.M6_Uhol_ToleranciaMIN.7:= P2_Srobovanie.PAR.M6_AtlasCopcoInputs[2].31;
    P2_Srobovanie.STAV.M6_Uhol_ToleranciaMIN.8:= P2_Srobovanie.PAR.M6_AtlasCopcoInputs[2].16;
    P2_Srobovanie.STAV.M6_Uhol_ToleranciaMIN.9:= P2_Srobovanie.PAR.M6_AtlasCopcoInputs[2].17;
    P2_Srobovanie.STAV.M6_Uhol_ToleranciaMIN.10:= P2_Srobovanie.PAR.M6_AtlasCopcoInputs[2].18;
    P2_Srobovanie.STAV.M6_Uhol_ToleranciaMIN.11:= P2_Srobovanie.PAR.M6_AtlasCopcoInputs[2].19;
    P2_Srobovanie.STAV.M6_Uhol_ToleranciaMIN.12:= P2_Srobovanie.PAR.M6_AtlasCopcoInputs[2].20;
    P2_Srobovanie.STAV.M6_Uhol_ToleranciaMIN.13:= P2_Srobovanie.PAR.M6_AtlasCopcoInputs[2].21;
    P2_Srobovanie.STAV.M6_Uhol_ToleranciaMIN.14:= P2_Srobovanie.PAR.M6_AtlasCopcoInputs[2].22;
    P2_Srobovanie.STAV.M6_Uhol_ToleranciaMIN.15:= P2_Srobovanie.PAR.M6_AtlasCopcoInputs[2].23;

END_ACTION
```

### Program Logical/Program/Pracovisko_2/P2_SkrutkovaciSet_M4 (IEC)

#### Main.st - Init, cyclic, exit code
```iecst
PROGRAM _INIT
    TprazdnyZasobnik.PT:=T#2000ms;
    TakumulaciaPlna.PT:=T#1000ms;
    TvytvorenieVakua.PT:=T#200ms;
    TodvetranieVakua.PT:=T#1s;
    TprefukPredBrzdou.PT:=T#2000ms;
    TprefukZaBrzdou.PT:=T#2000ms;
    TvysuvanieSpindle.PT:=T#1s;
    TpripravaSkrutky.PT:=T#3000ms;
    ToddelovacZakladnaPoloha.PT:=T#1000ms;
    TodsatieNecistot.PT:=T#1000ms;
    Tvibrovanie.PT:=T#3000ms;
    Stav_PodavacVycisteny:= FALSE;
    Stav_SkrutkaM4_Pripravena:= FALSE;
    TvyfukovaniePredVibrovanim.PT:= T#1000ms;
    TpodaniaSkrutky.PT:= T#1000ms;
    TpredSkrutkaPripravena.PT:= T#500ms;
    TvypnutieOfuku.PT:= T#2000ms;
    TalarmuVysunutiaSkrutkovacky.PT:= T#10s;
END_PROGRAM

PROGRAM _CYCLIC

    Cas_PresunuSkrutky.PT:= T#1M;
    Cas_PresunuSkrutky();

    (********************Mapovanie IN/OUT********************************)

    SkrutkovaciSet.Manual:= P2_Srobovanie.SkrutkovaciSet_M4.Manual;
    SkrutkovaciSet.Automat:= P2_Srobovanie.SkrutkovaciSet_M4.Automat;
    SkrutkovaciSet.SkrutkaOdobrata:=P2_Srobovanie.SkrutkovaciSet_M4.SkrutkaM4_Odobrata;
    P2_Srobovanie.SkrutkovaciSet_M4.SkrutkaM4_Pripravena:= SkrutkovaciSet.SkrutkaPripravena;
    P2_Srobovanie.SkrutkovaciSet_M4.CistenieUkoncene:= SkrutkovaciSet.CistenieVykonane;
    SkrutkovaciSet.VykonajCistenie:= P2_Srobovanie.SkrutkovaciSet_M4.Cistenie;

    SkrutkovaciSet.Vreteno.IN.BrakeClosed:=P2_Srobovanie.IN.SkrutkM4_Cist_BrzdaZatvoren_MS13;
    SkrutkovaciSet.Vreteno.IN.BrakeOpen:=P2_Srobovanie.IN.SkrutkM4_Cist_BrzdaOtvorena_MS12;
    SkrutkovaciSet.Vreteno.IN.DeptControl:=P2_Srobovanie.IN.SkrutkM4_ZASUNUTY_MS10;
    SkrutkovaciSet.Vreteno.IN.ScrewMeasurement:=P2_Srobovanie.IN.SkrutkM4_SrobaPresla_IS30;
    SkrutkovaciSet.Vreteno.IN.ScrewMeasurementBrake:=P2_Srobovanie.IN.SkrutkM4_Cist_SrobaPresla_IS35;

    IF P2_Srobovanie.SkrutkovaciSet_M4.Reset AND SkrutkovaciSet.VretenoFaza <> 102 AND SkrutkovaciSet.VretenoFaza <> 104 THEN
        SkrutkovaciSet.VretenoFaza:=0;
        P2_Srobovanie.SkrutkovaciSet_M4.Reset:= FALSE;
    END_IF

    SkrutkovaciSet.Zasobnik.IN.AccumulationSwitch:=P2_Srobovanie.IN.ZasobSrobM4_ListaPLNA_OS4;
    SkrutkovaciSet.Zasobnik.IN.FeederLevelControl:=P2_Srobovanie.IN.ZasobSrobM4_PRAZDNY_IS33;
    SkrutkovaciSet.Zasobnik.IN.ScrewMeasurement:=P2_Srobovanie.IN.NastrelSrobM4_SrobaPresla_IS34;

    P2_Srobovanie.OUT.SkrutkM4_Cist_OfukVakua_RUN_YV28:=SkrutkovaciSet.Vreteno.OUT.BlastAirBrake;
    P2_Srobovanie.OUT.SkrutkM4_Cist_OTVOR_YV27:=SkrutkovaciSet.Vreteno.OUT.BrakeSpindle;
    P2_Srobovanie.OUT.SkrutkM4_OfukVakua_RUN_YV25:=SkrutkovaciSet.Vreteno.OUT.CounterBlast;
    IF SkrutkovaciSet.VretenoFaza>1 AND SkrutkovaciSet.VretenoFaza<100 THEN
        P2_Srobovanie.OUT.SkrutkM4_VYSUN_YV24:=SkrutkovaciSet.Vreteno.OUT.Spindle;
    END_IF
    P2_Srobovanie.OUT.SkrutkM4_Cist_Vakum_RUN_YV29:=SkrutkovaciSet.Vreteno.OUT.WasteExtraction;
    IF SkrutkovaciSet.VykonajCistenie THEN
        P2_Srobovanie.OUT.SkrutkM4_PrisavSkrutky_RUN_YV26:=SkrutkovaciSet.Vreteno.OUT.Vacuum;
    END_IF
    P2_Srobovanie.OUT.ZasobSrobM4_Ofuk_RUN_YV20:=SkrutkovaciSet.Zasobnik.OUT.BlowOff;
    P2_Srobovanie.OUT.NastrelSrobM4_PosunSrobu_YV22:=SkrutkovaciSet.Zasobnik.OUT.Escapement;
    P2_Srobovanie.OUT.NastrelSrobM4_NastrelSrobu_YV23:=SkrutkovaciSet.Zasobnik.OUT.FeedAir;
    P2_Srobovanie.OUT.ZasobSrobM4_OfukTried_RUN_YV21:=SkrutkovaciSet.Zasobnik.OUT.SortingAir;
    P2_Srobovanie.OUT.ZasobSrobM4_Vibrovanie_RUN_FM3:= SkrutkovaciSet.Zasobnik.OUT.StartA20;
    (********************Časáky********************************)

    TprazdnyZasobnik();
    TakumulaciaPlna();
    TvytvorenieVakua();
    TodvetranieVakua();
    TprefukPredBrzdou();
    TprefukZaBrzdou();
    TvysuvanieSpindle();
    TpripravaSkrutky();
    ToddelovacZakladnaPoloha();
    TodsatieNecistot();
    Tvibrovanie();
    TvyfukovaniePredVibrovanim();
    TpodaniaSkrutky();
    TpredSkrutkaPripravena();
    TvypnutieOfuku();
    TalarmuVysunutiaSkrutkovacky();
    (********************Zásobnik********************************)

    //kontrola akumulacie
    IF SkrutkovaciSet.Zasobnik.IN.AccumulationSwitch=1 THEN
        TakumulaciaPlna.IN:=1;
    ELSE
        TakumulaciaPlna.IN:=0;
    END_IF

    //kontrola naplnenia zasobnika
    IF SkrutkovaciSet.Zasobnik.IN.FeederLevelControl=1 THEN
        TprazdnyZasobnik.IN:=1;
    ELSE
        TprazdnyZasobnik.IN:=0;
    END_IF

    //Ovládanie vzduchov zásobníka//
    IF ZapniHrniec THEN
        IF TakumulaciaPlna.Q=1 THEN
            SkrutkovaciSet.Zasobnik.OUT.BlowOff:=1;
        ELSE
            SkrutkovaciSet.Zasobnik.OUT.BlowOff:=0;
        END_IF
        SkrutkovaciSet.Zasobnik.OUT.SortingAir:= 1;
    ELSE
        SkrutkovaciSet.Zasobnik.OUT.BlowOff:=0;
    END_IF

    IF NOT SkrutkovaciSet.Zasobnik.OUT.StartA20 AND NOT ZapniHrniec THEN
        TvypnutieOfuku.IN:= 1;
    ELSE
        TvypnutieOfuku.IN:= 0;
    END_IF

    IF EDGEPOS(TvypnutieOfuku.Q) THEN
        SkrutkovaciSet.Zasobnik.OUT.SortingAir:= 0;
    END_IF

    //ovladanie vibracneho podavaca
    IF ZapniHrniec THEN
        TvyfukovaniePredVibrovanim.IN:= 1;
    ELSE
        TvyfukovaniePredVibrovanim.IN:= 0;
    END_IF

    IF ZapniHrniec AND TvyfukovaniePredVibrovanim.Q THEN
        SkrutkovaciSet.Zasobnik.OUT.StartA20:=1;
        Tvibrovanie.IN:=1;
    ELSE
        SkrutkovaciSet.Zasobnik.OUT.StartA20:=0;
        Tvibrovanie.IN:=0;
    END_IF

    IF Tvibrovanie.Q=1 THEN
        IF TakumulaciaPlna.Q=1 AND NOT P2_Srobovanie.RR_ZapniHrniec_M4 THEN
            ZapniHrniec:= 0;
        END_IF
    END_IF

    //Zapnutie hrnca v ručnom režime//
    IF EDGEPOS(P2_Srobovanie.RR_ZapniHrniec_M4) THEN
        ZapniHrniec:= TRUE;
    END_IF
    IF EDGENEG(P2_Srobovanie.RR_ZapniHrniec_M4) THEN
        ZapniHrniec:= FALSE;
    END_IF

    //Zrušenie signálu skrutka pripravená//
    IF SkrutkovaciSet.SkrutkaPripravena=1 THEN
        IF SkrutkovaciSet.SkrutkaOdobrata=1 THEN
            SkrutkovaciSet.SkrutkaPripravena:=0;
        END_IF
    END_IF

    (********************Vreteno********************************)
    CASE SkrutkovaciSet.VretenoFaza OF
        0: SkrutkovaciSet.VretenoStatus:="Vypnute";
            SkrutkovaciSet.Vreteno.OUT.BlastAirBrake:=0;
            SkrutkovaciSet.Vreteno.OUT.BrakeSpindle:=0;
            SkrutkovaciSet.Vreteno.OUT.CounterBlast:=0;
            SkrutkovaciSet.Vreteno.OUT.Spindle:=0;
            SkrutkovaciSet.Vreteno.OUT.Vacuum:=0;
            SkrutkovaciSet.Vreteno.OUT.WasteExtraction:=0;

            SkrutkovaciSet.Zasobnik.OUT.Escapement:=0;
            SkrutkovaciSet.Zasobnik.OUT.FeedAir:=0;

            SkrutkovaciSet.Zasobnik.OUT.StartA20:=0;

            SkrutkovaciSet.CistenieVykonane:=0;
            SkrutkovaciSet.SkrutkaPripravena:=0;

            TprazdnyZasobnik.IN:=0;
            TakumulaciaPlna.IN:=0;
            TvytvorenieVakua.IN:=0;
            TodvetranieVakua.IN:=0;
            TprefukPredBrzdou.IN:=0;
            TprefukZaBrzdou.IN:=0;
            TvysuvanieSpindle.IN:=0;
            TpripravaSkrutky.IN:=0;
            ToddelovacZakladnaPoloha.IN:=0;
            TodsatieNecistot.IN:=0;
            TpodaniaSkrutky.IN:= 0;
            TpredSkrutkaPripravena.IN:= 0;
            ZapniHrniec:= 0;
            PocetPokusovOpripravuSkrutky:=0;
            StavSkrutkovackaVysunuta:= 0;
            TalarmuVysunutiaSkrutkovacky.IN:= 0;
            SkrutkovaciSet.VretenoFaza:=1;

        1: SkrutkovaciSet.VretenoStatus:="Inicializacia: cakam na povel";
            IF SkrutkovaciSet.Automat=1 THEN
                SkrutkovaciSet.CistenieVykonane:=0;
                SkrutkovaciSet.SkrutkaPripravena:=0;
                SkrutkovaciSet.VretenoFaza:=2;
            ELSIF SkrutkovaciSet.Manual=1 THEN
                SkrutkovaciSet.VretenoFaza:=250;
            END_IF

        2: SkrutkovaciSet.VretenoStatus:="Inicializacia: cakam na povel precisti hadice";

            IF SkrutkovaciSet.VykonajCistenie=1 THEN
                SkrutkovaciSet.Vreteno.OUT.Vacuum:=1;
                SkrutkovaciSet.VretenoFaza:=3;
            END_IF

        3: SkrutkovaciSet.VretenoStatus:="Inicializacia: Cakam na snimac: vreteno vysunute";
            SkrutkovaciSet.Vreteno.OUT.Spindle:=1;
            TalarmuVysunutiaSkrutkovacky.IN:= 1;

            IF P2_Srobovanie.IN.SkrutkM4_VysunutieHrotu_IOS4 > 1 THEN
                StavSkrutkovackaVysunuta:= TRUE;
                TvysuvanieSpindle.IN:=1;
            END_IF

            IF TvysuvanieSpindle.Q=1 AND StavSkrutkovackaVysunuta THEN
                TodvetranieVakua.IN:= 1;
                SkrutkovaciSet.Vreteno.OUT.CounterBlast:=1;
                SkrutkovaciSet.Vreteno.OUT.Vacuum:=0;
            END_IF

            IF TvysuvanieSpindle.Q AND StavSkrutkovackaVysunuta AND TodvetranieVakua.Q THEN
                StavSkrutkovackaVysunuta:= FALSE;
                TalarmuVysunutiaSkrutkovacky.IN:= 0;
                TvysuvanieSpindle.IN:=0;
                TodvetranieVakua.IN:= 0;
                SkrutkovaciSet.VretenoFaza:=4;
            ELSIF TalarmuVysunutiaSkrutkovacky.Q THEN
                P2_Alarmy[268]:= TRUE;
                P2_PoruchaST3:= TRUE;
            END_IF

        4: SkrutkovaciSet.VretenoStatus:="Inicializacia: Cakam na snimac: vreteno zasunute";
            SkrutkovaciSet.Vreteno.OUT.Spindle:=0;
            IF SkrutkovaciSet.Vreteno.IN.DeptControl=1 THEN
                SkrutkovaciSet.Vreteno.OUT.CounterBlast:=0;
                SkrutkovaciSet.VretenoFaza:=5;
            END_IF

        5: SkrutkovaciSet.VretenoStatus:="Inicializacia: Cakam na prefuknutie hadice za brzdou";
            TprefukZaBrzdou.IN:=1;
            SkrutkovaciSet.Vreteno.OUT.BlastAirBrake:=1;
            IF TprefukZaBrzdou.Q=1 THEN
                TprefukZaBrzdou.IN:=0;
                SkrutkovaciSet.Vreteno.OUT.BlastAirBrake:=0;
                SkrutkovaciSet.VretenoFaza:=6;
            END_IF

        6: SkrutkovaciSet.VretenoStatus:="Inicializacia: vypinam prefuk";
            TprefukZaBrzdou.IN:=0;
            SkrutkovaciSet.Vreteno.OUT.BlastAirBrake:=0;
            SkrutkovaciSet.Vreteno.OUT.Vacuum:=1;
            SkrutkovaciSet.VretenoFaza:=7;

        7: SkrutkovaciSet.VretenoStatus:="Inicializacia: Cakam na snimac: vreteno vysunute";
            SkrutkovaciSet.Vreteno.OUT.Spindle:=1;
            TalarmuVysunutiaSkrutkovacky.IN:= 1;

            IF P2_Srobovanie.IN.SkrutkM4_VysunutieHrotu_IOS4 > 1 THEN
                StavSkrutkovackaVysunuta:= TRUE;
                TvysuvanieSpindle.IN:=1;
            END_IF

            IF TvysuvanieSpindle.Q=1 AND StavSkrutkovackaVysunuta THEN
                TodvetranieVakua.IN:= 1;
                SkrutkovaciSet.Vreteno.OUT.CounterBlast:=1;
                SkrutkovaciSet.Vreteno.OUT.Vacuum:=0;
            END_IF

            IF TvysuvanieSpindle.Q AND StavSkrutkovackaVysunuta AND TodvetranieVakua.Q THEN
                StavSkrutkovackaVysunuta:= FALSE;
                TalarmuVysunutiaSkrutkovacky.IN:= 0;
                TvysuvanieSpindle.IN:=0;
                TodvetranieVakua.IN:= 0;
                SkrutkovaciSet.VretenoFaza:=8;
            ELSIF TalarmuVysunutiaSkrutkovacky.Q THEN
                P2_Alarmy[268]:= TRUE;
                P2_PoruchaST3:= TRUE;
            END_IF

        8: SkrutkovaciSet.VretenoStatus:="Inicializacia: Cakam na snimac: vreteno zasunute";
            SkrutkovaciSet.Vreteno.OUT.Spindle:=0;
            IF SkrutkovaciSet.Vreteno.IN.DeptControl=1 THEN
                SkrutkovaciSet.Vreteno.OUT.CounterBlast:=0;
                SkrutkovaciSet.VretenoFaza:=9;
            END_IF

        9: SkrutkovaciSet.VretenoStatus:="Inicializacia: Cakam na prefuknutie hadice pred brzdou";
            TprefukPredBrzdou.IN:=1;
            SkrutkovaciSet.Zasobnik.OUT.FeedAir:=1;
            IF TprefukPredBrzdou.Q=1 THEN
                TprefukPredBrzdou.IN:=0;
                SkrutkovaciSet.Zasobnik.OUT.FeedAir:=0;
                SkrutkovaciSet.VretenoFaza:=10;
            END_IF

        10: SkrutkovaciSet.VretenoStatus:="Inicializacia: Cakam na snimac: brzda uvolnena";
            SkrutkovaciSet.Vreteno.OUT.BrakeSpindle:=1;
            IF SkrutkovaciSet.Vreteno.IN.BrakeOpen=1 THEN
                SkrutkovaciSet.Vreteno.OUT.BlastAirBrake:=1;
                SkrutkovaciSet.VretenoFaza:=11;
            END_IF

        11: SkrutkovaciSet.VretenoStatus:="Inicializacia: Cakam na prefuknutie hadice za brzdou";
            TprefukZaBrzdou.IN:=1;
            SkrutkovaciSet.Vreteno.OUT.BlastAirBrake:=1;
            IF TprefukZaBrzdou.Q=1 THEN
                TprefukZaBrzdou.IN:=0;
                SkrutkovaciSet.Vreteno.OUT.BlastAirBrake:=0;
                SkrutkovaciSet.VretenoFaza:=12;
            END_IF

        12: SkrutkovaciSet.VretenoStatus:="Inicializacia: vypinam prefuk";
            TprefukZaBrzdou.IN:=0;
            SkrutkovaciSet.Vreteno.OUT.BlastAirBrake:=0;
            SkrutkovaciSet.Vreteno.OUT.Vacuum:=1;
            SkrutkovaciSet.VretenoFaza:=13;

        13: SkrutkovaciSet.VretenoStatus:="Inicializacia: Cakam na snimac: vreteno vysunute";
            SkrutkovaciSet.Vreteno.OUT.Spindle:=1;
            TalarmuVysunutiaSkrutkovacky.IN:= 1;

            IF P2_Srobovanie.IN.SkrutkM4_VysunutieHrotu_IOS4 > 1 THEN
                StavSkrutkovackaVysunuta:= TRUE;
                TvysuvanieSpindle.IN:=1;
            END_IF

            IF TvysuvanieSpindle.Q=1 AND StavSkrutkovackaVysunuta THEN
                TodvetranieVakua.IN:= 1;
                SkrutkovaciSet.Vreteno.OUT.CounterBlast:=1;
                SkrutkovaciSet.Vreteno.OUT.Vacuum:=0;
            END_IF

            IF TvysuvanieSpindle.Q AND StavSkrutkovackaVysunuta AND TodvetranieVakua.Q THEN
                StavSkrutkovackaVysunuta:= FALSE;
                TalarmuVysunutiaSkrutkovacky.IN:= 0;
                TvysuvanieSpindle.IN:=0;
                TodvetranieVakua.IN:= 0;
                SkrutkovaciSet.VretenoFaza:=14;
            ELSIF TalarmuVysunutiaSkrutkovacky.Q THEN
                P2_Alarmy[268]:= TRUE;
                P2_PoruchaST3:= TRUE;
            END_IF

        14: SkrutkovaciSet.VretenoStatus:="Inicializacia: Cakam na snimac: vreteno zasunute";
            SkrutkovaciSet.Vreteno.OUT.Spindle:=0;
            IF SkrutkovaciSet.Vreteno.IN.DeptControl=1 THEN
                SkrutkovaciSet.Vreteno.OUT.CounterBlast:=0;
                SkrutkovaciSet.VretenoFaza:=15;
            END_IF

        15: SkrutkovaciSet.VretenoStatus:="Inicializacia: Cakam na snimac: brzda zasunuta";
            SkrutkovaciSet.Vreteno.OUT.BrakeSpindle:=0;
            IF SkrutkovaciSet.Vreteno.IN.BrakeClosed=1 THEN
                SkrutkovaciSet.CistenieVykonane:=1;
                SkrutkovaciSet.VretenoFaza:=16;
            END_IF

        16: SkrutkovaciSet.VretenoStatus:="Inicializacia: Cakam na zrusenie signalu: vykonaj cistenie";
            IF SkrutkovaciSet.VykonajCistenie=0 THEN
                SkrutkovaciSet.CistenieVykonane:=0;
                SkrutkovaciSet.SkrutkaPripravena:=0;
                SkrutkovaciSet.VretenoFaza:=100;
            END_IF

        100: SkrutkovaciSet.VretenoStatus:="Cakam kym zasobnik pripravy skrutku";
            ZapniHrniec:= 1;
            IF TakumulaciaPlna.Q=1 AND SkrutkovaciSet.Zasobnik.OUT.StartA20 THEN
                TpodaniaSkrutky.IN:= 1;
            END_IF

            IF TpodaniaSkrutky.Q THEN
                TpodaniaSkrutky.IN:= 0;
                SkrutkovaciSet.VretenoFaza:=102;
            END_IF

        102: SkrutkovaciSet.VretenoStatus:="Cakam na snimac: skrutka presla hadicou";
            SkrutkovaciSet.Zasobnik.OUT.Escapement:=1;
            Cas_PresunuSkrutky.IN:= TRUE;
            TpripravaSkrutky.IN:=1;
            IF SkrutkovaciSet.Zasobnik.IN.ScrewMeasurement=1 THEN
                SkrutkovaciSet.Zasobnik.OUT.FeedAir:=1;
                TpripravaSkrutky.IN:=0;
                NameranyCasPresunuSkrutky:= Cas_PresunuSkrutky.ET;
                Cas_PresunuSkrutky.IN:= FALSE;
                SkrutkovaciSet.VretenoFaza:=104;
            ELSIF TpripravaSkrutky.Q=1 THEN
                Cas_PresunuSkrutky.IN:= FALSE;
                TpripravaSkrutky.IN:=0;
                SkrutkovaciSet.Zasobnik.OUT.Escapement:=0;
                SkrutkovaciSet.VretenoFaza:=100;
            END_IF

        104: SkrutkovaciSet.VretenoStatus:="Cakam na snimac: skrutka presla hadicou pred brzdou";
            IF SkrutkovaciSet.Vreteno.IN.ScrewMeasurementBrake=1 THEN
                SkrutkovaciSet.Zasobnik.OUT.Escapement:=0;
                SkrutkovaciSet.Zasobnik.OUT.FeedAir:=0;
                PocetPokusovOpripravuSkrutky:=0;
                SkrutkovaciSet.VretenoFaza:=106;
            END_IF

        106: SkrutkovaciSet.VretenoStatus:="Cakam na odsatie necistot";
            SkrutkovaciSet.Vreteno.OUT.WasteExtraction:=1;
            TodsatieNecistot.IN:=1;

            IF TodsatieNecistot.Q=1 THEN
                TodsatieNecistot.IN:=0;
                SkrutkovaciSet.Vreteno.OUT.WasteExtraction:=0;
                SkrutkovaciSet.VretenoFaza:=107;
            END_IF

        107: SkrutkovaciSet.VretenoStatus:="Cakam kym skrutkovacka odoberie skrutku";
            IF SkrutkovaciSet.SkrutkaPripravena=0 AND SkrutkovaciSet.SkrutkaOdobrata=0 THEN
                SkrutkovaciSet.VretenoFaza:=108;
            END_IF

        108: SkrutkovaciSet.VretenoStatus:="Cakam na snimac: brzda uvolnena";
            SkrutkovaciSet.Vreteno.OUT.BrakeSpindle:=1;
            IF SkrutkovaciSet.Vreteno.IN.BrakeOpen=1 THEN
                SkrutkovaciSet.Vreteno.OUT.BlastAirBrake:=1;
                SkrutkovaciSet.VretenoFaza:=110;
            END_IF

        110: SkrutkovaciSet.VretenoStatus:="Cakam na snimac: skrutka presla hadicou pred vretenom";
            IF SkrutkovaciSet.Vreteno.IN.ScrewMeasurement=1 THEN
                SkrutkovaciSet.Vreteno.OUT.BlastAirBrake:=0;
                SkrutkovaciSet.Vreteno.OUT.BrakeSpindle:=0;
                SkrutkovaciSet.VretenoFaza:=112;
            END_IF

        112: SkrutkovaciSet.VretenoStatus:="Cakam na snimac: brzda zabrzdena";
            SkrutkovaciSet.Vreteno.OUT.BrakeSpindle:=0;
            IF SkrutkovaciSet.Vreteno.IN.BrakeClosed=1 AND SkrutkovaciSet.SkrutkaOdobrata=0 THEN
                TpredSkrutkaPripravena.IN:= 1;
                IF TpredSkrutkaPripravena.Q THEN
                    TpredSkrutkaPripravena.IN:= 0;
                    SkrutkovaciSet.SkrutkaPripravena:=1;
                    SkrutkovaciSet.VretenoFaza:=100;
                END_IF
            END_IF

            //*************** opakovany pokus o oddelenie skrutky *********************************

        170: SkrutkovaciSet.VretenoStatus:="Cakam na presunutie oddelovaca do zakladnej polohy";
            SkrutkovaciSet.Zasobnik.OUT.Escapement:=0;
            ToddelovacZakladnaPoloha.IN:=1;
            IF ToddelovacZakladnaPoloha.Q=1 THEN
                ToddelovacZakladnaPoloha.IN:=0;
                PocetPokusovOpripravuSkrutky:=PocetPokusovOpripravuSkrutky+1;
                IF PocetPokusovOpripravuSkrutky>3 THEN
                    PocetPokusovOpripravuSkrutky:=0;
                    SkrutkovaciSet.VretenoFaza:=171;
                ELSE
                    SkrutkovaciSet.VretenoFaza:=100;
                END_IF
            END_IF

        171: SkrutkovaciSet.VretenoStatus:="Zaseknuta skrutka v oddelovaci!!!";
    END_CASE

END_PROGRAM

PROGRAM _EXIT
	(* Insert code here *)

END_PROGRAM
```

#### Types.typ - Local data types
```iecst
TYPE
	SkrutkovaciSetStruc : 	STRUCT
		VretenoStatus : WSTRING[80];
		VretenoFaza : USINT;
		Zasobnik : ZasobnikStruc;
		Vreteno : VretenoStruc;
		SkrutkaOdobrata : BOOL;
		SkrutkaPripravena : BOOL;
		Manual : BOOL;
		PodajSrobu : BOOL;
		CistenieVykonane : BOOL;
		VykonajCistenie : BOOL;
		Automat : BOOL;
	END_STRUCT;
	INzasobnik : 	STRUCT
		AccumulationSwitch : BOOL; (*Snimac zaplnenia S25*)
		ScrewMeasurement : BOOL; (*Kontrola matice S21*)
		FeederLevelControl : BOOL; (*Hladina v zasobniku S20*)
	END_STRUCT;
	OUTzasobnik : 	STRUCT
		StartA20 : BOOL; (*Zapnutie vibrovania A20*)
		Escapement : BOOL; (*Pustanie matky do hadice Y22*)
		FeedAir : BOOL; (*Strielanie do hadice Y21*)
		SortingAir : BOOL; (*Triedenie kusov Y30*)
		BlowOff : BOOL; (*Zhadzovanie kusov Y25*)
	END_STRUCT;
	INvreteno : 	STRUCT
		ReturnStroke : BOOL; (*Vreteno zasunute S01*)
		DeptControl : BOOL; (*Vreteno vysunute S02*)
		BrakeClosed : BOOL; (*Brzda zatvorena S13*)
		BrakeOpen : BOOL; (*Brzda otvorena S12*)
		ScrewMeasurementBrake : BOOL; (*Kontrola matice pred brzdou S15*)
		ScrewMeasurement : BOOL; (*Kontrola matice v hadici S06*)
	END_STRUCT;
	OUTvreteno : 	STRUCT
		WasteExtraction : BOOL; (*Odstranovanie spiny Y13*)
		Spindle : BOOL; (*Vysunutie vretena Y02*)
		BlastAirBrake : BOOL; (*Strielanie za brzdou Y14*)
		BrakeSpindle : BOOL; (*Brzda vretena Y12*)
		Vacuum : BOOL; (*Pridrzanie skrutky Y15*)
		CounterBlast : BOOL; (*Uvolnenie skrutky Y16*)
	END_STRUCT;
	VretenoStruc : 	STRUCT
		OUT : OUTvreteno;
		IN : INvreteno;
	END_STRUCT;
	ZasobnikStruc : 	STRUCT
		OUT : OUTzasobnik;
		IN : INzasobnik;
	END_STRUCT;
END_TYPE
```

#### Variables.var - Local variables
```iecst
VAR
	Stav_PodavacVycisteny : BOOL;
	Stav_SkrutkaM4_Pripravena : BOOL;
	SkrutkovaciSet : SkrutkovaciSetStruc;
	TprazdnyZasobnik : TON;
	TakumulaciaPlna : TON;
	TvytvorenieVakua : TON;
	TodvetranieVakua : TON;
	TprefukPredBrzdou : TON;
	TvysuvanieSpindle : TON;
	TprefukZaBrzdou : TON;
	PocetPokusovOpripravuSkrutky : USINT;
	ToddelovacZakladnaPoloha : TON;
	TpripravaSkrutky : TON;
	TodsatieNecistot : TON;
	Tvibrovanie : TON;
	TvyfukovaniePredVibrovanim : TON;
	ZapniHrniec : BOOL;
	TpodaniaSkrutky : TON;
	TpredSkrutkaPripravena : TON;
	TvypnutieOfuku : TON;
	StavSkrutkovackaVysunuta : BOOL;
	TalarmuVysunutiaSkrutkovacky : TON;
END_VAR
```

### Program Logical/Program/Pracovisko_2/P2_SkrutkovaciSet_M5 (IEC)

#### Main.st - Init, cyclic, exit code
```iecst
PROGRAM _INIT
    TprazdnyZasobnik.PT:=T#2000ms;
    TakumulaciaPlna.PT:=T#3000ms;
    TvytvorenieVakua.PT:=T#200ms;
    TodvetranieVakua.PT:=T#1s;
    TprefukPredBrzdou.PT:=T#2000ms;
    TprefukZaBrzdou.PT:=T#2000ms;
    TvysuvanieSpindle.PT:=T#1s;
    TpripravaSkrutky.PT:=T#3000ms;
    ToddelovacZakladnaPoloha.PT:=T#1000ms;
    TodsatieNecistot.PT:=T#1000ms;
    Tvibrovanie.PT:=T#12000ms;
    Stav_PodavacVycisteny:= FALSE;
    Stav_SkrutkaM5_Pripravena:= FALSE;
    TvyfukovaniePredVibrovanim.PT:= T#1000ms;
    TpodaniaSkrutky.PT:= T#1000ms;
    TpredSkrutkaPripravena.PT:= T#100ms;
    TvypnutieOfuku.PT:= T#2000ms;
    TalarmuVysunutiaSkrutkovacky.PT:= T#10s;
END_PROGRAM

PROGRAM _CYCLIC

   (********************Mapovanie IN/OUT********************************)

    SkrutkovaciSet.Manual:= P2_Srobovanie.SkrutkovaciSet_M5.Manual;
    SkrutkovaciSet.Automat:= P2_Srobovanie.SkrutkovaciSet_M5.Automat;
    SkrutkovaciSet.SkrutkaOdobrata:=P2_Srobovanie.SkrutkovaciSet_M5.SkrutkaM5_Odobrata;
    P2_Srobovanie.SkrutkovaciSet_M5.SkrutkaM5_Pripravena:= SkrutkovaciSet.SkrutkaPripravena;
    P2_Srobovanie.SkrutkovaciSet_M5.CistenieUkoncene:= SkrutkovaciSet.CistenieVykonane;
    SkrutkovaciSet.VykonajCistenie:= P2_Srobovanie.SkrutkovaciSet_M5.Cistenie;

    SkrutkovaciSet.Vreteno.IN.BrakeClosed:=P2_Srobovanie.IN.SkrutkM5_Cist_BrzdaZatvorena_MS2;
    SkrutkovaciSet.Vreteno.IN.BrakeOpen:=P2_Srobovanie.IN.SkrutkM5_Cist_BrzdaOtvorena_MS1;
    SkrutkovaciSet.Vreteno.IN.DeptControl:=P2_Srobovanie.IN.SkrutkM5_ZASUNUTY_MS11;
    SkrutkovaciSet.Vreteno.IN.ScrewMeasurement:=P2_Srobovanie.IN.SkrutkM5_SrobaPresla_IS32;
    SkrutkovaciSet.Vreteno.IN.ScrewMeasurementBrake:=P2_Srobovanie.IN.SkrutkM5_Cist_SrobaPresla_IS31;

    IF P2_Srobovanie.SkrutkovaciSet_M5.Reset AND SkrutkovaciSet.VretenoFaza <> 102 AND SkrutkovaciSet.VretenoFaza <> 104 THEN
        SkrutkovaciSet.VretenoFaza:=0;
        P2_Srobovanie.SkrutkovaciSet_M5.Reset:= FALSE;
    END_IF

    SkrutkovaciSet.Zasobnik.IN.AccumulationSwitch:=P2_Srobovanie.IN.ZasobSrobM5_ListaPLNA_OS3;
    SkrutkovaciSet.Zasobnik.IN.FeederLevelControl:=P2_Srobovanie.IN.ZasobSrobM5_PRAZDNY_IS28;
    SkrutkovaciSet.Zasobnik.IN.ScrewMeasurement:=P2_Srobovanie.IN.NastrelSrobM5_SrobaPresla_IS29;

    P2_Srobovanie.OUT.SkrutkM5_Cist_OfukVakua_RUN_YV17:=SkrutkovaciSet.Vreteno.OUT.BlastAirBrake;
    P2_Srobovanie.OUT.SkrutkM5_Cist_OTVOR_YV19:=SkrutkovaciSet.Vreteno.OUT.BrakeSpindle;
    P2_Srobovanie.OUT.SkrutkM5_OfukVakua_RUN_YV15:=SkrutkovaciSet.Vreteno.OUT.CounterBlast;
    IF SkrutkovaciSet.VretenoFaza>1 AND SkrutkovaciSet.VretenoFaza<100 THEN
        P2_Srobovanie.OUT.SkrutkM5_VYSUN_YV14:=SkrutkovaciSet.Vreteno.OUT.Spindle;
    END_IF
    P2_Srobovanie.OUT.SkrutkM5_Cist_Vakum_RUN_YV18:=SkrutkovaciSet.Vreteno.OUT.WasteExtraction;
    IF SkrutkovaciSet.VykonajCistenie THEN
        P2_Srobovanie.OUT.SkrutkM5_PrisavSkrutky_RUN_YV16:=SkrutkovaciSet.Vreteno.OUT.Vacuum;
    END_IF
    P2_Srobovanie.OUT.ZasobSrobM5_Ofuk_RUN_YV10:=SkrutkovaciSet.Zasobnik.OUT.BlowOff;
    P2_Srobovanie.OUT.NastrelSrobM5_PosunSrobu_YV12:=SkrutkovaciSet.Zasobnik.OUT.Escapement;
    P2_Srobovanie.OUT.NastrelSrobM5_NastrelSrobu_YV13:=SkrutkovaciSet.Zasobnik.OUT.FeedAir;
    P2_Srobovanie.OUT.ZasobSrobM5_OfukTried_RUN_YV11:=SkrutkovaciSet.Zasobnik.OUT.SortingAir;
    P2_Srobovanie.OUT.ZasobSrobM5_Vibrovanie_RUN_FM4:= SkrutkovaciSet.Zasobnik.OUT.StartA20;

    (********************Časáky********************************)
    TprazdnyZasobnik();
    TakumulaciaPlna();
    TvytvorenieVakua();
    TodvetranieVakua();
    TprefukPredBrzdou();
    TprefukZaBrzdou();
    TvysuvanieSpindle();
    TpripravaSkrutky();
    ToddelovacZakladnaPoloha();
    TodsatieNecistot();
    Tvibrovanie();
    TvyfukovaniePredVibrovanim();
    TpodaniaSkrutky();
    TpredSkrutkaPripravena();
    TvypnutieOfuku();
    TalarmuVysunutiaSkrutkovacky();
    (********************Zásobnik********************************)

    //kontrola akumulacie
    IF SkrutkovaciSet.Zasobnik.IN.AccumulationSwitch=1 THEN
        TakumulaciaPlna.IN:=1;
    ELSE
        TakumulaciaPlna.IN:=0;
    END_IF

    //kontrola naplnenia zasobnika
    IF SkrutkovaciSet.Zasobnik.IN.FeederLevelControl=1 THEN
        TprazdnyZasobnik.IN:=1;
    ELSE
        TprazdnyZasobnik.IN:=0;
    END_IF

    //Ovládanie vzduchov zásobníka//
    IF ZapniHrniec THEN
        IF TakumulaciaPlna.Q=1 THEN
            SkrutkovaciSet.Zasobnik.OUT.BlowOff:=1;
        ELSE
            SkrutkovaciSet.Zasobnik.OUT.BlowOff:=0;
        END_IF
        SkrutkovaciSet.Zasobnik.OUT.SortingAir:= 1;
    ELSE
        SkrutkovaciSet.Zasobnik.OUT.BlowOff:=0;
    END_IF

    IF NOT SkrutkovaciSet.Zasobnik.OUT.StartA20 AND NOT ZapniHrniec THEN
        TvypnutieOfuku.IN:= 1;
    ELSE
        TvypnutieOfuku.IN:= 0;
    END_IF

    IF EDGEPOS(TvypnutieOfuku.Q)  THEN
        SkrutkovaciSet.Zasobnik.OUT.SortingAir:= 0;
    END_IF

    //ovladanie vibracneho podavaca
    IF ZapniHrniec THEN
        TvyfukovaniePredVibrovanim.IN:= 1;
    ELSE
        TvyfukovaniePredVibrovanim.IN:= 0;
    END_IF

    IF ZapniHrniec AND TvyfukovaniePredVibrovanim.Q THEN
        SkrutkovaciSet.Zasobnik.OUT.StartA20:=1;
        Tvibrovanie.IN:=1;
    ELSE
        SkrutkovaciSet.Zasobnik.OUT.StartA20:=0;
        Tvibrovanie.IN:=0;
    END_IF

    IF Tvibrovanie.Q=1 THEN
        IF TakumulaciaPlna.Q=1 AND NOT P2_Srobovanie.RR_ZapniHrniec_M5 THEN
            ZapniHrniec:= 0;
        END_IF
    END_IF

    //Zapnutie hrnca v ručnom režime//
    IF EDGEPOS(P2_Srobovanie.RR_ZapniHrniec_M5) THEN
        ZapniHrniec:= TRUE;
    END_IF
    IF EDGENEG(P2_Srobovanie.RR_ZapniHrniec_M5) THEN
        ZapniHrniec:= FALSE;
    END_IF

    //Zrušenie signálu skrutka pripravená//
    IF SkrutkovaciSet.SkrutkaPripravena=1 THEN
        IF SkrutkovaciSet.SkrutkaOdobrata=1 THEN
            SkrutkovaciSet.SkrutkaPripravena:=0;
        END_IF
    END_IF

    (********************Vreteno********************************)
    CASE SkrutkovaciSet.VretenoFaza OF
        0: SkrutkovaciSet.VretenoStatus:="Vypnute";
            SkrutkovaciSet.Vreteno.OUT.BlastAirBrake:=0;
            SkrutkovaciSet.Vreteno.OUT.BrakeSpindle:=0;
            SkrutkovaciSet.Vreteno.OUT.CounterBlast:=0;
            SkrutkovaciSet.Vreteno.OUT.Spindle:=0;
            SkrutkovaciSet.Vreteno.OUT.Vacuum:=0;
            SkrutkovaciSet.Vreteno.OUT.WasteExtraction:=0;

            SkrutkovaciSet.Zasobnik.OUT.Escapement:=0;
            SkrutkovaciSet.Zasobnik.OUT.FeedAir:=0;

            SkrutkovaciSet.Zasobnik.OUT.StartA20:=0;

            SkrutkovaciSet.CistenieVykonane:=0;
            SkrutkovaciSet.SkrutkaPripravena:=0;

            TprazdnyZasobnik.IN:=0;
            TakumulaciaPlna.IN:=0;
            TvytvorenieVakua.IN:=0;
            TodvetranieVakua.IN:=0;
            TprefukPredBrzdou.IN:=0;
            TprefukZaBrzdou.IN:=0;
            TvysuvanieSpindle.IN:=0;
            TpripravaSkrutky.IN:=0;
            ToddelovacZakladnaPoloha.IN:=0;
            TodsatieNecistot.IN:=0;
            TpodaniaSkrutky.IN:= 0;
            TpredSkrutkaPripravena.IN:= 0;
            ZapniHrniec:= 0;
            PocetPokusovOpripravuSkrutky:=0;
            StavSkrutkovackaVysunuta:= 0;
            TalarmuVysunutiaSkrutkovacky.IN:= 0;
            SkrutkovaciSet.VretenoFaza:=1;

        1: SkrutkovaciSet.VretenoStatus:="Inicializacia: cakam na povel";
            IF SkrutkovaciSet.Automat=1 THEN
                SkrutkovaciSet.CistenieVykonane:=0;
                SkrutkovaciSet.SkrutkaPripravena:=0;
                SkrutkovaciSet.VretenoFaza:=2;
            ELSIF SkrutkovaciSet.Manual=1 THEN
                SkrutkovaciSet.VretenoFaza:=250;
            END_IF

        2: SkrutkovaciSet.VretenoStatus:="Inicializacia: cakam na povel precisti hadice";

            IF SkrutkovaciSet.VykonajCistenie=1 THEN
                SkrutkovaciSet.Vreteno.OUT.Vacuum:=1;
                SkrutkovaciSet.VretenoFaza:=3;
            END_IF

        3: SkrutkovaciSet.VretenoStatus:="Inicializacia: Cakam na snimac: vreteno vysunute";
            SkrutkovaciSet.Vreteno.OUT.Spindle:=1;
            TalarmuVysunutiaSkrutkovacky.IN:= 1;

            IF P2_Srobovanie.IN.SkrutkM5_VysunutieHrotu_IOS5 > 1 THEN
                StavSkrutkovackaVysunuta:= TRUE;
                TvysuvanieSpindle.IN:=1;
            END_IF

            IF TvysuvanieSpindle.Q=1 AND StavSkrutkovackaVysunuta THEN
                TodvetranieVakua.IN:= 1;
                SkrutkovaciSet.Vreteno.OUT.CounterBlast:=1;
                SkrutkovaciSet.Vreteno.OUT.Vacuum:=0;
            END_IF

            IF TvysuvanieSpindle.Q AND StavSkrutkovackaVysunuta AND TodvetranieVakua.Q THEN
                StavSkrutkovackaVysunuta:= FALSE;
                TalarmuVysunutiaSkrutkovacky.IN:= 0;
                TvysuvanieSpindle.IN:=0;
                TodvetranieVakua.IN:= 0;
                SkrutkovaciSet.VretenoFaza:=4;
            ELSIF TalarmuVysunutiaSkrutkovacky.Q THEN
                P2_Alarmy[269]:= TRUE;
                P2_PoruchaST3:= TRUE;
            END_IF

        4: SkrutkovaciSet.VretenoStatus:="Inicializacia: Cakam na snimac: vreteno zasunute";
            SkrutkovaciSet.Vreteno.OUT.Spindle:=0;
            IF SkrutkovaciSet.Vreteno.IN.DeptControl=1 THEN
                SkrutkovaciSet.Vreteno.OUT.CounterBlast:=0;
                SkrutkovaciSet.VretenoFaza:=5;
            END_IF

        5: SkrutkovaciSet.VretenoStatus:="Inicializacia: Cakam na prefuknutie hadice za brzdou";
            TprefukZaBrzdou.IN:=1;
            SkrutkovaciSet.Vreteno.OUT.BlastAirBrake:=1;
            IF TprefukZaBrzdou.Q=1 THEN
                TprefukZaBrzdou.IN:=0;
                SkrutkovaciSet.Vreteno.OUT.BlastAirBrake:=0;
                SkrutkovaciSet.VretenoFaza:=6;
            END_IF

        6: SkrutkovaciSet.VretenoStatus:="Inicializacia: vypinam prefuk";
            TprefukZaBrzdou.IN:=0;
            SkrutkovaciSet.Vreteno.OUT.BlastAirBrake:=0;
            SkrutkovaciSet.Vreteno.OUT.Vacuum:=1;
            SkrutkovaciSet.VretenoFaza:=7;

        7: SkrutkovaciSet.VretenoStatus:="Inicializacia: Cakam na snimac: vreteno vysunute";
            SkrutkovaciSet.Vreteno.OUT.Spindle:=1;
            TalarmuVysunutiaSkrutkovacky.IN:= 1;

            IF P2_Srobovanie.IN.SkrutkM5_VysunutieHrotu_IOS5 > 1 THEN
                StavSkrutkovackaVysunuta:= TRUE;
                TvysuvanieSpindle.IN:=1;
            END_IF

            IF TvysuvanieSpindle.Q=1 AND StavSkrutkovackaVysunuta THEN
                TodvetranieVakua.IN:= 1;
                SkrutkovaciSet.Vreteno.OUT.CounterBlast:=1;
                SkrutkovaciSet.Vreteno.OUT.Vacuum:=0;
            END_IF

            IF TvysuvanieSpindle.Q AND StavSkrutkovackaVysunuta AND TodvetranieVakua.Q THEN
                StavSkrutkovackaVysunuta:= FALSE;
                TalarmuVysunutiaSkrutkovacky.IN:= 0;
                TvysuvanieSpindle.IN:=0;
                TodvetranieVakua.IN:= 0;
                SkrutkovaciSet.VretenoFaza:=8;
            ELSIF TalarmuVysunutiaSkrutkovacky.Q THEN
                P2_Alarmy[269]:= TRUE;
                P2_PoruchaST3:= TRUE;
            END_IF

        8: SkrutkovaciSet.VretenoStatus:="Inicializacia: Cakam na snimac: vreteno zasunute";
            SkrutkovaciSet.Vreteno.OUT.Spindle:=0;
            IF SkrutkovaciSet.Vreteno.IN.DeptControl=1 THEN
                SkrutkovaciSet.Vreteno.OUT.CounterBlast:=0;
                SkrutkovaciSet.VretenoFaza:=9;
            END_IF

        9: SkrutkovaciSet.VretenoStatus:="Inicializacia: Cakam na prefuknutie hadice pred brzdou";
            TprefukPredBrzdou.IN:=1;
            SkrutkovaciSet.Zasobnik.OUT.FeedAir:=1;
            IF TprefukPredBrzdou.Q=1 THEN
                TprefukPredBrzdou.IN:=0;
                SkrutkovaciSet.Zasobnik.OUT.FeedAir:=0;
                SkrutkovaciSet.VretenoFaza:=10;
            END_IF

        10: SkrutkovaciSet.VretenoStatus:="Inicializacia: Cakam na snimac: brzda uvolnena";
            SkrutkovaciSet.Vreteno.OUT.BrakeSpindle:=1;
            IF SkrutkovaciSet.Vreteno.IN.BrakeOpen=1 THEN
                SkrutkovaciSet.Vreteno.OUT.BlastAirBrake:=1;
                SkrutkovaciSet.VretenoFaza:=11;
            END_IF

        11: SkrutkovaciSet.VretenoStatus:="Inicializacia: Cakam na prefuknutie hadice za brzdou";
            TprefukZaBrzdou.IN:=1;
            SkrutkovaciSet.Vreteno.OUT.BlastAirBrake:=1;
            IF TprefukZaBrzdou.Q=1 THEN
                TprefukZaBrzdou.IN:=0;
                SkrutkovaciSet.Vreteno.OUT.BlastAirBrake:=0;
                SkrutkovaciSet.VretenoFaza:=12;
            END_IF

        12: SkrutkovaciSet.VretenoStatus:="Inicializacia: vypinam prefuk";
            TprefukZaBrzdou.IN:=0;
            SkrutkovaciSet.Vreteno.OUT.BlastAirBrake:=0;
            SkrutkovaciSet.Vreteno.OUT.Vacuum:=1;
            SkrutkovaciSet.VretenoFaza:=13;

        13: SkrutkovaciSet.VretenoStatus:="Inicializacia: Cakam na snimac: vreteno vysunute";
            SkrutkovaciSet.Vreteno.OUT.Spindle:=1;
            TalarmuVysunutiaSkrutkovacky.IN:= 1;

            IF P2_Srobovanie.IN.SkrutkM5_VysunutieHrotu_IOS5 > 1 THEN
                StavSkrutkovackaVysunuta:= TRUE;
                TvysuvanieSpindle.IN:=1;
            END_IF

            IF TvysuvanieSpindle.Q=1 AND StavSkrutkovackaVysunuta THEN
                TodvetranieVakua.IN:= 1;
                SkrutkovaciSet.Vreteno.OUT.CounterBlast:=1;
                SkrutkovaciSet.Vreteno.OUT.Vacuum:=0;
            END_IF

            IF TvysuvanieSpindle.Q AND StavSkrutkovackaVysunuta AND TodvetranieVakua.Q THEN
                StavSkrutkovackaVysunuta:= FALSE;
                TalarmuVysunutiaSkrutkovacky.IN:= 0;
                TvysuvanieSpindle.IN:=0;
                TodvetranieVakua.IN:= 0;
                SkrutkovaciSet.VretenoFaza:=14;
            ELSIF TalarmuVysunutiaSkrutkovacky.Q THEN
                P2_Alarmy[269]:= TRUE;
                P2_PoruchaST3:= TRUE;
            END_IF

        14: SkrutkovaciSet.VretenoStatus:="Inicializacia: Cakam na snimac: vreteno zasunute";
            SkrutkovaciSet.Vreteno.OUT.Spindle:=0;
            IF SkrutkovaciSet.Vreteno.IN.DeptControl=1 THEN
                SkrutkovaciSet.Vreteno.OUT.CounterBlast:=0;
                SkrutkovaciSet.VretenoFaza:=15;
            END_IF

        15: SkrutkovaciSet.VretenoStatus:="Inicializacia: Cakam na snimac: brzda zasunuta";
            SkrutkovaciSet.Vreteno.OUT.BrakeSpindle:=0;
            IF SkrutkovaciSet.Vreteno.IN.BrakeClosed=1 THEN
                SkrutkovaciSet.CistenieVykonane:=1;
                SkrutkovaciSet.VretenoFaza:=16;
            END_IF

        16: SkrutkovaciSet.VretenoStatus:="Inicializacia: Cakam na zrusenie signalu: vykonaj cistenie";
            IF SkrutkovaciSet.VykonajCistenie=0 THEN
                SkrutkovaciSet.CistenieVykonane:=0;
                SkrutkovaciSet.SkrutkaPripravena:=0;
                SkrutkovaciSet.VretenoFaza:=100;
            END_IF

        100: SkrutkovaciSet.VretenoStatus:="Cakam kym zasobnik pripravy skrutku";
            ZapniHrniec:= 1;
            IF TakumulaciaPlna.Q=1 AND SkrutkovaciSet.Zasobnik.OUT.StartA20 THEN
                TpodaniaSkrutky.IN:= 1;
            END_IF

            IF TpodaniaSkrutky.Q THEN
                TpodaniaSkrutky.IN:= 0;
                SkrutkovaciSet.VretenoFaza:=102;
            END_IF

        102: SkrutkovaciSet.VretenoStatus:="Cakam na snimac: skrutka presla hadicou";
            SkrutkovaciSet.Zasobnik.OUT.Escapement:=1;
            TpripravaSkrutky.IN:=1;
            IF SkrutkovaciSet.Zasobnik.IN.ScrewMeasurement=1 THEN
                SkrutkovaciSet.Zasobnik.OUT.FeedAir:=1;
                TpripravaSkrutky.IN:=0;
                SkrutkovaciSet.VretenoFaza:=104;
            ELSIF TpripravaSkrutky.Q=1 THEN
                TpripravaSkrutky.IN:=0;
                SkrutkovaciSet.Zasobnik.OUT.Escapement:=0;
                SkrutkovaciSet.VretenoFaza:=100;
            END_IF

        104: SkrutkovaciSet.VretenoStatus:="Cakam na snimac: skrutka presla hadicou pred brzdou";
            IF SkrutkovaciSet.Vreteno.IN.ScrewMeasurementBrake=1 THEN
                SkrutkovaciSet.Zasobnik.OUT.Escapement:=0;
                SkrutkovaciSet.Zasobnik.OUT.FeedAir:=0;
                PocetPokusovOpripravuSkrutky:=0;
                SkrutkovaciSet.VretenoFaza:=106;
            END_IF

        106: SkrutkovaciSet.VretenoStatus:="Cakam na odsatie necistot";
            SkrutkovaciSet.Vreteno.OUT.WasteExtraction:=1;
            TodsatieNecistot.IN:=1;

            IF TodsatieNecistot.Q=1 THEN
                TodsatieNecistot.IN:=0;
                SkrutkovaciSet.Vreteno.OUT.WasteExtraction:=0;
                SkrutkovaciSet.VretenoFaza:=107;
            END_IF

        107: SkrutkovaciSet.VretenoStatus:="Cakam kym skrutkovacka odoberie skrutku";
            IF SkrutkovaciSet.SkrutkaPripravena=0 AND SkrutkovaciSet.SkrutkaOdobrata=0 THEN
                SkrutkovaciSet.VretenoFaza:=108;
            END_IF

        108: SkrutkovaciSet.VretenoStatus:="Cakam na snimac: brzda uvolnena";
            SkrutkovaciSet.Vreteno.OUT.BrakeSpindle:=1;
            IF SkrutkovaciSet.Vreteno.IN.BrakeOpen=1 THEN
                SkrutkovaciSet.Vreteno.OUT.BlastAirBrake:=1;
                SkrutkovaciSet.VretenoFaza:=110;
            END_IF

        110: SkrutkovaciSet.VretenoStatus:="Cakam na snimac: skrutka presla hadicou pred vretenom";
            IF SkrutkovaciSet.Vreteno.IN.ScrewMeasurement=1 THEN
                SkrutkovaciSet.Vreteno.OUT.BlastAirBrake:=0;
                SkrutkovaciSet.Vreteno.OUT.BrakeSpindle:=0;
                SkrutkovaciSet.VretenoFaza:=112;
            END_IF

        112: SkrutkovaciSet.VretenoStatus:="Cakam na snimac: brzda zabrzdena";
            SkrutkovaciSet.Vreteno.OUT.BrakeSpindle:=0;
            IF SkrutkovaciSet.Vreteno.IN.BrakeClosed=1 AND SkrutkovaciSet.SkrutkaOdobrata=0 THEN
                TpredSkrutkaPripravena.IN:= 1;
                IF TpredSkrutkaPripravena.Q THEN
                    TpredSkrutkaPripravena.IN:= 0;
                    SkrutkovaciSet.SkrutkaPripravena:=1;
                    SkrutkovaciSet.VretenoFaza:=100;
                END_IF
            END_IF

            //*************** opakovany pokus o oddelenie skrutky *********************************

        170: SkrutkovaciSet.VretenoStatus:="Cakam na presunutie oddelovaca do zakladnej polohy";
            SkrutkovaciSet.Zasobnik.OUT.Escapement:=0;
            ToddelovacZakladnaPoloha.IN:=1;
            IF ToddelovacZakladnaPoloha.Q=1 THEN
                ToddelovacZakladnaPoloha.IN:=0;
                PocetPokusovOpripravuSkrutky:=PocetPokusovOpripravuSkrutky+1;
                IF PocetPokusovOpripravuSkrutky>3 THEN
                    PocetPokusovOpripravuSkrutky:=0;
                    SkrutkovaciSet.VretenoFaza:=171;
                ELSE
                    SkrutkovaciSet.VretenoFaza:=100;
                END_IF
            END_IF

        171: SkrutkovaciSet.VretenoStatus:="Zaseknuta skrutka v oddelovaci!!!";
    END_CASE

END_PROGRAM

PROGRAM _EXIT
	(* Insert code here *)

END_PROGRAM
```
